      A(    ;
      A     M   2000.6;
      AN    M   2001.0;
      A     M   2010.4;
      A     M   2201.0;
      O     ;
      A     M   2000.5;
      A     DB51.DBX  608.4;
      A     DB51.DBX  603.7;
      AN    DB51.DBX  603.6;
      O     M   2001.2;
      )     ;
      A     M   2204.3;
      A     M   2208.7;
      AN    M   2204.1;
      AN    M   2242.0;
      =     M   2242.1;
NETWORK
TITLE =

      A(    ;
      A     M   2000.6;
      AN    M   2001.0;
      AN    M   2010.4;
      A     M   2201.0;
      O     ;
      A     M   2000.5;
      A     DB51.DBX  608.5;
      A     DB51.DBX  603.6;
      AN    DB51.DBX  603.7;
      )     ;
      A     M   2204.0;
      A     M   2208.7;
      AN    M   2204.2;
      AN    M   2242.3;
      =     M   2242.2;
NETWORK
TITLE =

      A(    ;
      A     M   2000.6;
      AN    M   2001.0;
      A     M   2010.4;
      A     M   2201.0;
      O     ;
      A     M   2000.5;
      A     DB51.DBX  608.5;
      A     DB51.DBX  603.7;
      AN    DB51.DBX  603.6;
      O     M   2001.2;
      )     ;
      A     M   2204.0;
      A     M   2208.7;
      AN    M   2204.3;
      AN    M   2242.2;
      =     M   2242.3;
NETWORK
TITLE =
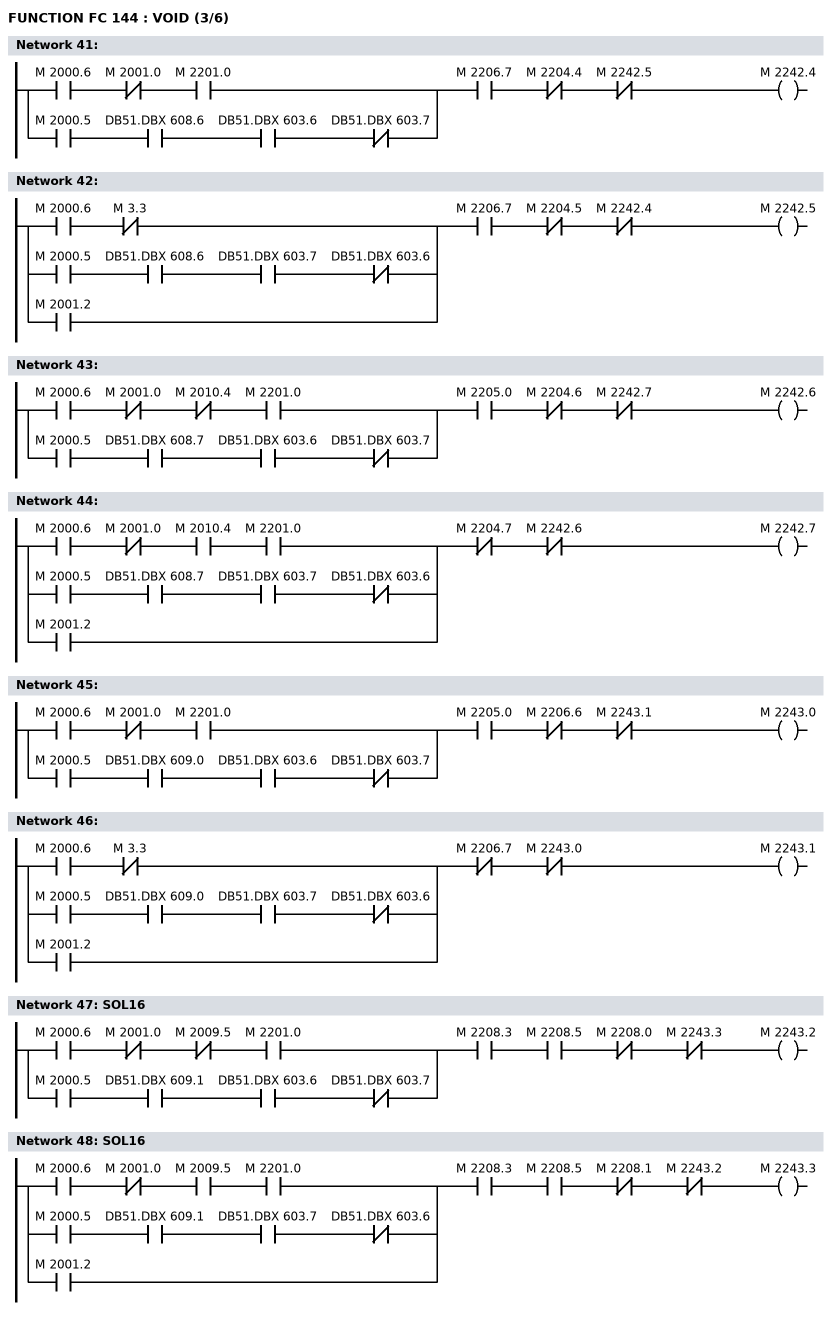

      A(    ;
      A     M   2000.6;
      AN    M   2001.0;
      A     M   2201.0;
      O     ;
      A     M   2000.5;
      A     DB51.DBX  608.6;
      A     DB51.DBX  603.6;
      AN    DB51.DBX  603.7;
      )     ;
      A     M   2206.7;
      AN    M   2204.4;
      AN    M   2242.5;
      =     M   2242.4;
NETWORK
TITLE =

      A(    ;
      A     M   2000.6;
      AN    M      3.3;
      O     ;
      A     M   2000.5;
      A     DB51.DBX  608.6;
      A     DB51.DBX  603.7;
      AN    DB51.DBX  603.6;
      O     M   2001.2;
      )     ;
      A     M   2206.7;
      AN    M   2204.5;
      AN    M   2242.4;
      =     M   2242.5;
NETWORK
TITLE =

      A(    ;
      A     M   2000.6;
      AN    M   2001.0;
      AN    M   2010.4;
      A     M   2201.0;
      O     ;
      A     M   2000.5;
      A     DB51.DBX  608.7;
      A     DB51.DBX  603.6;
      AN    DB51.DBX  603.7;
      )     ;
      A     M   2205.0;
      AN    M   2204.6;
      AN    M   2242.7;
      =     M   2242.6;
NETWORK
TITLE =

      A(    ;
      A     M   2000.6;
      AN    M   2001.0;
      A     M   2010.4;
      A     M   2201.0;
      O     ;
      A     M   2000.5;
      A     DB51.DBX  608.7;
      A     DB51.DBX  603.7;
      AN    DB51.DBX  603.6;
      O     M   2001.2;
      )     ;
      AN    M   2204.7;
      AN    M   2242.6;
      =     M   2242.7;
NETWORK
TITLE =

      A(    ;
      A     M   2000.6;
      AN    M   2001.0;
      A     M   2201.0;
      O     ;
      A     M   2000.5;
      A     DB51.DBX  609.0;
      A     DB51.DBX  603.6;
      AN    DB51.DBX  603.7;
      )     ;
      A     M   2205.0;
      AN    M   2206.6;
      AN    M   2243.1;
      =     M   2243.0;
NETWORK
TITLE =

      A(    ;
      A     M   2000.6;
      AN    M      3.3;
      O     ;
      A     M   2000.5;
      A     DB51.DBX  609.0;
      A     DB51.DBX  603.7;
      AN    DB51.DBX  603.6;
      O     M   2001.2;
      )     ;
      AN    M   2206.7;
      AN    M   2243.0;
      =     M   2243.1;
NETWORK
TITLE =SOL16

      A(    ;
      A     M   2000.6;
      AN    M   2001.0;
      AN    M   2009.5;
      A     M   2201.0;
      O     ;
      A     M   2000.5;
      A     DB51.DBX  609.1;
      A     DB51.DBX  603.6;
      AN    DB51.DBX  603.7;
      )     ;
      A     M   2208.3;
      A     M   2208.5;
      AN    M   2208.0;
      AN    M   2243.3;
      =     M   2243.2;
NETWORK
TITLE =SOL16

      A(    ;
      A     M   2000.6;
      AN    M   2001.0;
      A     M   2009.5;
      A     M   2201.0;
      O     ;
      A     M   2000.5;
      A     DB51.DBX  609.1;
      A     DB51.DBX  603.7;
      AN    DB51.DBX  603.6;
      O     M   2001.2;
      )     ;
      A     M   2208.3;
      A     M   2208.5;
      AN    M   2208.1;
      AN    M   2243.2;
      =     M   2243.3;
NETWORK
TITLE =SOL17
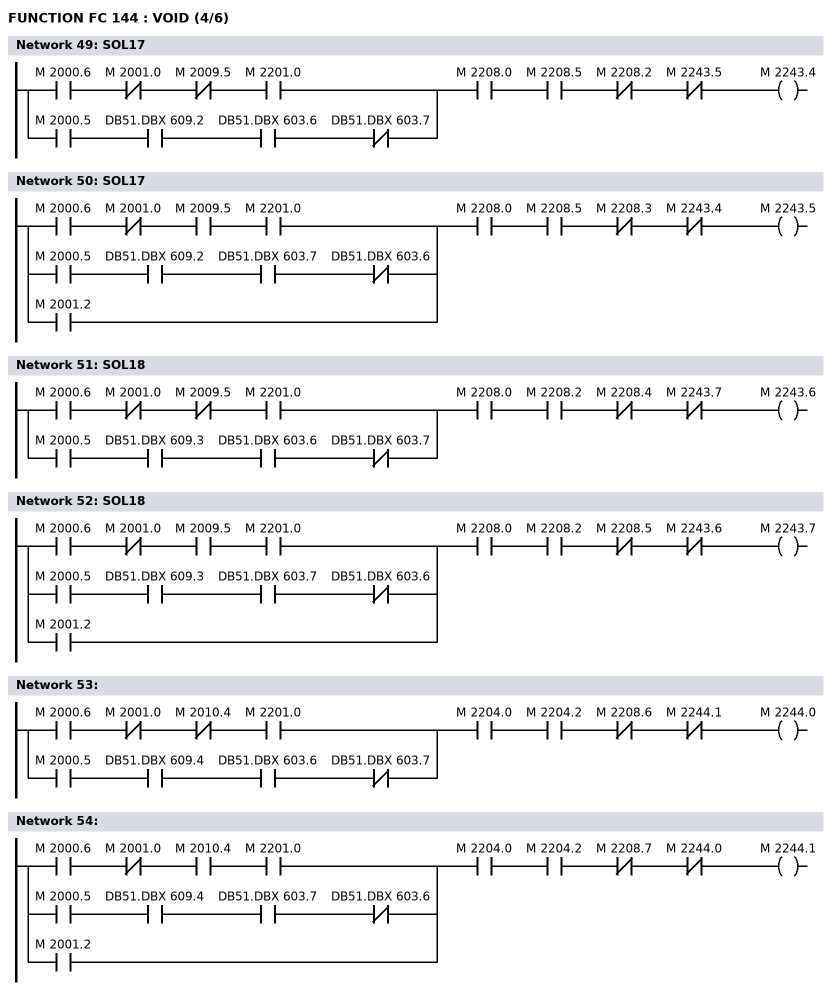

      A(    ;
      A     M   2000.6;
      AN    M   2001.0;
      AN    M   2009.5;
      A     M   2201.0;
      O     ;
      A     M   2000.5;
      A     DB51.DBX  609.2;
      A     DB51.DBX  603.6;
      AN    DB51.DBX  603.7;
      )     ;
      A     M   2208.0;
      A     M   2208.5;
      AN    M   2208.2;
      AN    M   2243.5;
      =     M   2243.4;
NETWORK
TITLE =SOL17

      A(    ;
      A     M   2000.6;
      AN    M   2001.0;
      A     M   2009.5;
      A     M   2201.0;
      O     ;
      A     M   2000.5;
      A     DB51.DBX  609.2;
      A     DB51.DBX  603.7;
      AN    DB51.DBX  603.6;
      O     M   2001.2;
      )     ;
      A     M   2208.0;
      A     M   2208.5;
      AN    M   2208.3;
      AN    M   2243.4;
      =     M   2243.5;
NETWORK
TITLE =SOL18

      A(    ;
      A     M   2000.6;
      AN    M   2001.0;
      AN    M   2009.5;
      A     M   2201.0;
      O     ;
      A     M   2000.5;
      A     DB51.DBX  609.3;
      A     DB51.DBX  603.6;
      AN    DB51.DBX  603.7;
      )     ;
      A     M   2208.0;
      A     M   2208.2;
      AN    M   2208.4;
      AN    M   2243.7;
      =     M   2243.6;
NETWORK
TITLE =SOL18

      A(    ;
      A     M   2000.6;
      AN    M   2001.0;
      A     M   2009.5;
      A     M   2201.0;
      O     ;
      A     M   2000.5;
      A     DB51.DBX  609.3;
      A     DB51.DBX  603.7;
      AN    DB51.DBX  603.6;
      O     M   2001.2;
      )     ;
      A     M   2208.0;
      A     M   2208.2;
      AN    M   2208.5;
      AN    M   2243.6;
      =     M   2243.7;
NETWORK
TITLE =

      A(    ;
      A     M   2000.6;
      AN    M   2001.0;
      AN    M   2010.4;
      A     M   2201.0;
      O     ;
      A     M   2000.5;
      A     DB51.DBX  609.4;
      A     DB51.DBX  603.6;
      AN    DB51.DBX  603.7;
      )     ;
      A     M   2204.0;
      A     M   2204.2;
      AN    M   2208.6;
      AN    M   2244.1;
      =     M   2244.0;
NETWORK
TITLE =

      A(    ;
      A     M   2000.6;
      AN    M   2001.0;
      A     M   2010.4;
      A     M   2201.0;
      O     ;
      A     M   2000.5;
      A     DB51.DBX  609.4;
      A     DB51.DBX  603.7;
      AN    DB51.DBX  603.6;
      O     M   2001.2;
      )     ;
      A     M   2204.0;
      A     M   2204.2;
      AN    M   2208.7;
      AN    M   2244.0;
      =     M   2244.1;
NETWORK
TITLE =TL 대차 SOL 동작회로
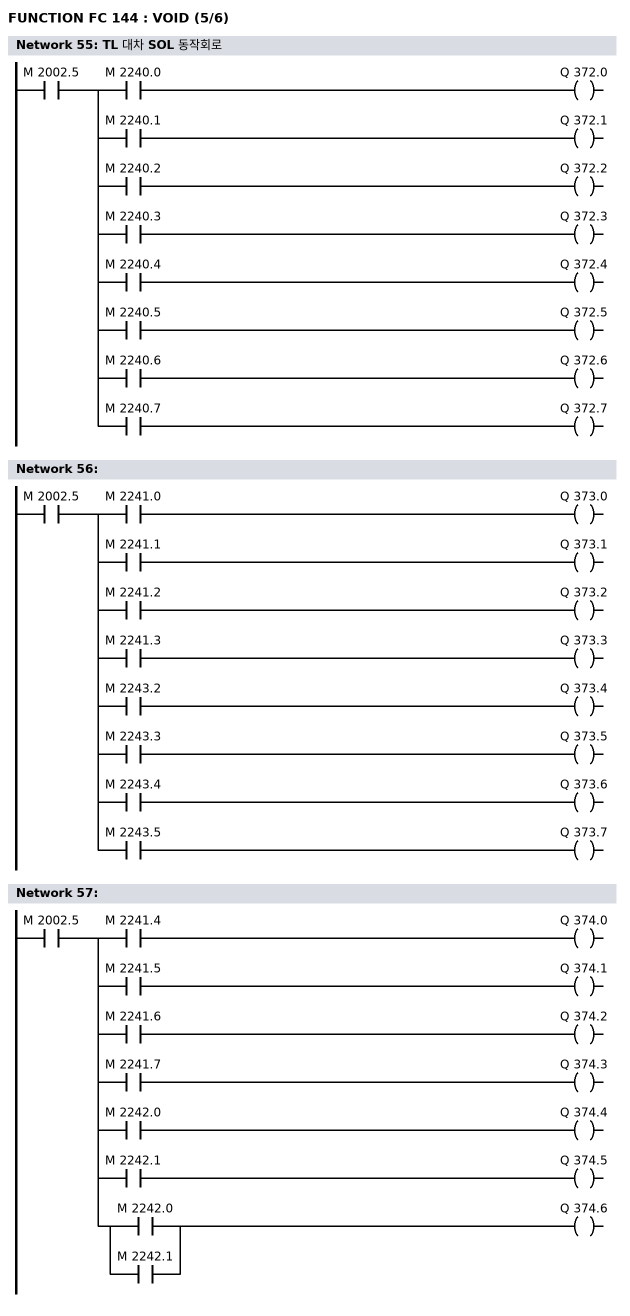

      A     M   2002.5;
      =     L      0.0;
      A     L      0.0;
      A     M   2240.0;
      =     Q    372.0;
      A     L      0.0;
      A     M   2240.1;
      =     Q    372.1;
      A     L      0.0;
      A     M   2240.2;
      =     Q    372.2;
      A     L      0.0;
      A     M   2240.3;
      =     Q    372.3;
      A     L      0.0;
      A     M   2240.4;
      =     Q    372.4;
      A     L      0.0;
      A     M   2240.5;
      =     Q    372.5;
      A     L      0.0;
      A     M   2240.6;
      =     Q    372.6;
      A     L      0.0;
      A     M   2240.7;
      =     Q    372.7;
NETWORK
TITLE =

      A     M   2002.5;
      =     L      0.0;
      A     L      0.0;
      A     M   2241.0;
      =     Q    373.0;
      A     L      0.0;
      A     M   2241.1;
      =     Q    373.1;
      A     L      0.0;
      A     M   2241.2;
      =     Q    373.2;
      A     L      0.0;
      A     M   2241.3;
      =     Q    373.3;
      A     L      0.0;
      A     M   2243.2;
      =     Q    373.4;
      A     L      0.0;
      A     M   2243.3;
      =     Q    373.5;
      A     L      0.0;
      A     M   2243.4;
      =     Q    373.6;
      A     L      0.0;
      A     M   2243.5;
      =     Q    373.7;
NETWORK
TITLE =

      A     M   2002.5;
      =     L      0.0;
      A     L      0.0;
      A     M   2241.4;
      =     Q    374.0;
      A     L      0.0;
      A     M   2241.5;
      =     Q    374.1;
      A     L      0.0;
      A     M   2241.6;
      =     Q    374.2;
      A     L      0.0;
      A     M   2241.7;
      =     Q    374.3;
      A     L      0.0;
      A     M   2242.0;
      =     Q    374.4;
      A     L      0.0;
      A     M   2242.1;
      =     Q    374.5;
      A     L      0.0;
      A(    ;
      O     M   2242.0;
      O     M   2242.1;
      )     ;
      =     Q    374.6;
NETWORK
TITLE =
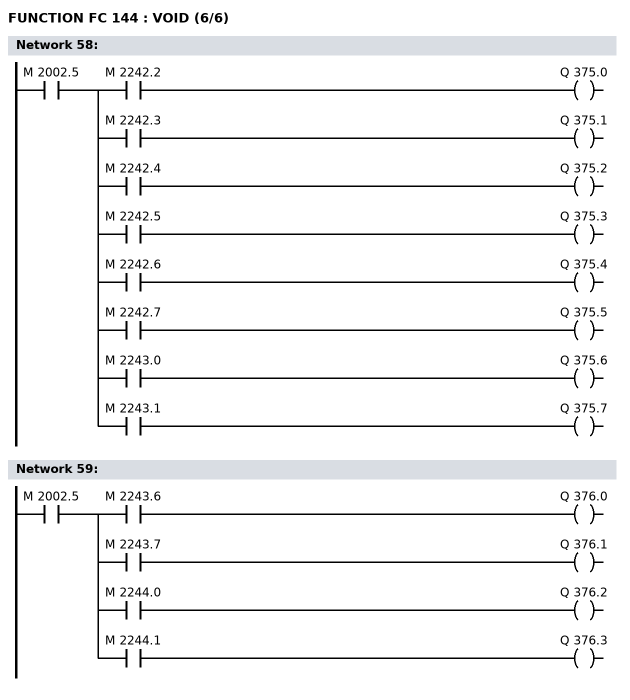

      A     M   2002.5;
      =     L      0.0;
      A     L      0.0;
      A     M   2242.2;
      =     Q    375.0;
      A     L      0.0;
      A     M   2242.3;
      =     Q    375.1;
      A     L      0.0;
      A     M   2242.4;
      =     Q    375.2;
      A     L      0.0;
      A     M   2242.5;
      =     Q    375.3;
      A     L      0.0;
      A     M   2242.6;
      =     Q    375.4;
      A     L      0.0;
      A     M   2242.7;
      =     Q    375.5;
      A     L      0.0;
      A     M   2243.0;
      =     Q    375.6;
      A     L      0.0;
      A     M   2243.1;
      =     Q    375.7;
NETWORK
TITLE =

      A     M   2002.5;
      =     L      0.0;
      A     L      0.0;
      A     M   2243.6;
      =     Q    376.0;
      A     L      0.0;
      A     M   2243.7;
      =     Q    376.1;
      A     L      0.0;
      A     M   2244.0;
      =     Q    376.2;
      A     L      0.0;
      A     M   2244.1;
      =     Q    376.3;
END_FUNCTION

FUNCTION FC 145 : VOID
TITLE =
VERSION : 0.1

BEGIN
NETWORK
TITLE =
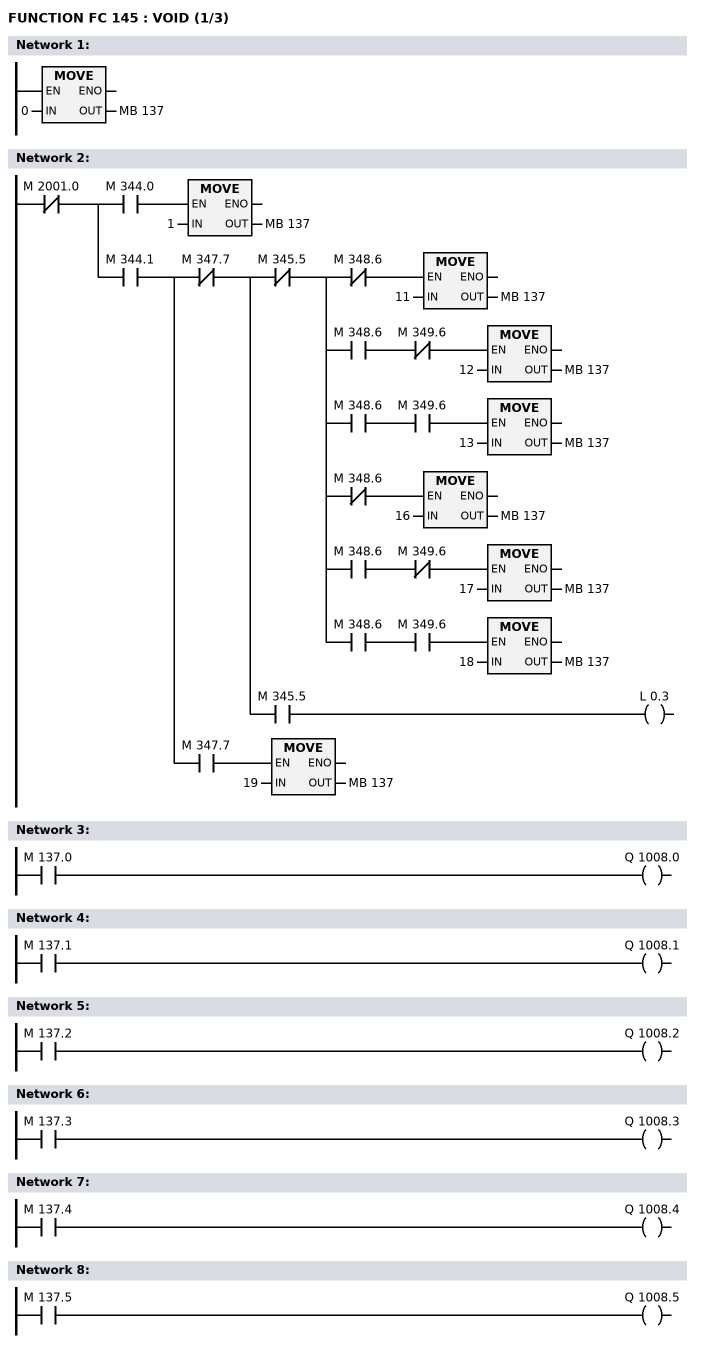

      L     0;
      T     MB   137;
      NOP   0;
NETWORK
TITLE =

      AN    M   2001.0;
      =     L      0.0;
      A     L      0.0;
      A     M    344.0;
      JNB   _001;
      L     1;
      T     MB   137;
_001: NOP   0;
      A     L      0.0;
      A     M    344.1;
      =     L      0.1;
      A     L      0.1;
      AN    M    347.7;
      =     L      0.2;
      A     L      0.2;
      AN    M    345.5;
      =     L      0.3;
      A     L      0.3;
      AN    M    348.6;
      JNB   _002;
      L     11;
      T     MB   137;
_002: NOP   0;
      A     L      0.3;
      A     M    348.6;
      AN    M    349.6;
      JNB   _003;
      L     12;
      T     MB   137;
_003: NOP   0;
      A     L      0.3;
      A     M    348.6;
      A     M    349.6;
      JNB   _004;
      L     13;
      T     MB   137;
_004: NOP   0;
      A     L      0.2;
      A     M    345.5;
      =     L      0.3;
      A     L      0.3;
      AN    M    348.6;
      JNB   _005;
      L     16;
      T     MB   137;
_005: NOP   0;
      A     L      0.3;
      A     M    348.6;
      AN    M    349.6;
      JNB   _006;
      L     17;
      T     MB   137;
_006: NOP   0;
      A     L      0.3;
      A     M    348.6;
      A     M    349.6;
      JNB   _007;
      L     18;
      T     MB   137;
_007: NOP   0;
      A     L      0.1;
      A     M    347.7;
      JNB   _008;
      L     19;
      T     MB   137;
_008: NOP   0;
NETWORK
TITLE =

      A     M    137.0;
      =     Q   1008.0;
NETWORK
TITLE =

      A     M    137.1;
      =     Q   1008.1;
NETWORK
TITLE =

      A     M    137.2;
      =     Q   1008.2;
NETWORK
TITLE =

      A     M    137.3;
      =     Q   1008.3;
NETWORK
TITLE =

      A     M    137.4;
      =     Q   1008.4;
NETWORK
TITLE =

      A     M    137.5;
      =     Q   1008.5;
NETWORK
TITLE =
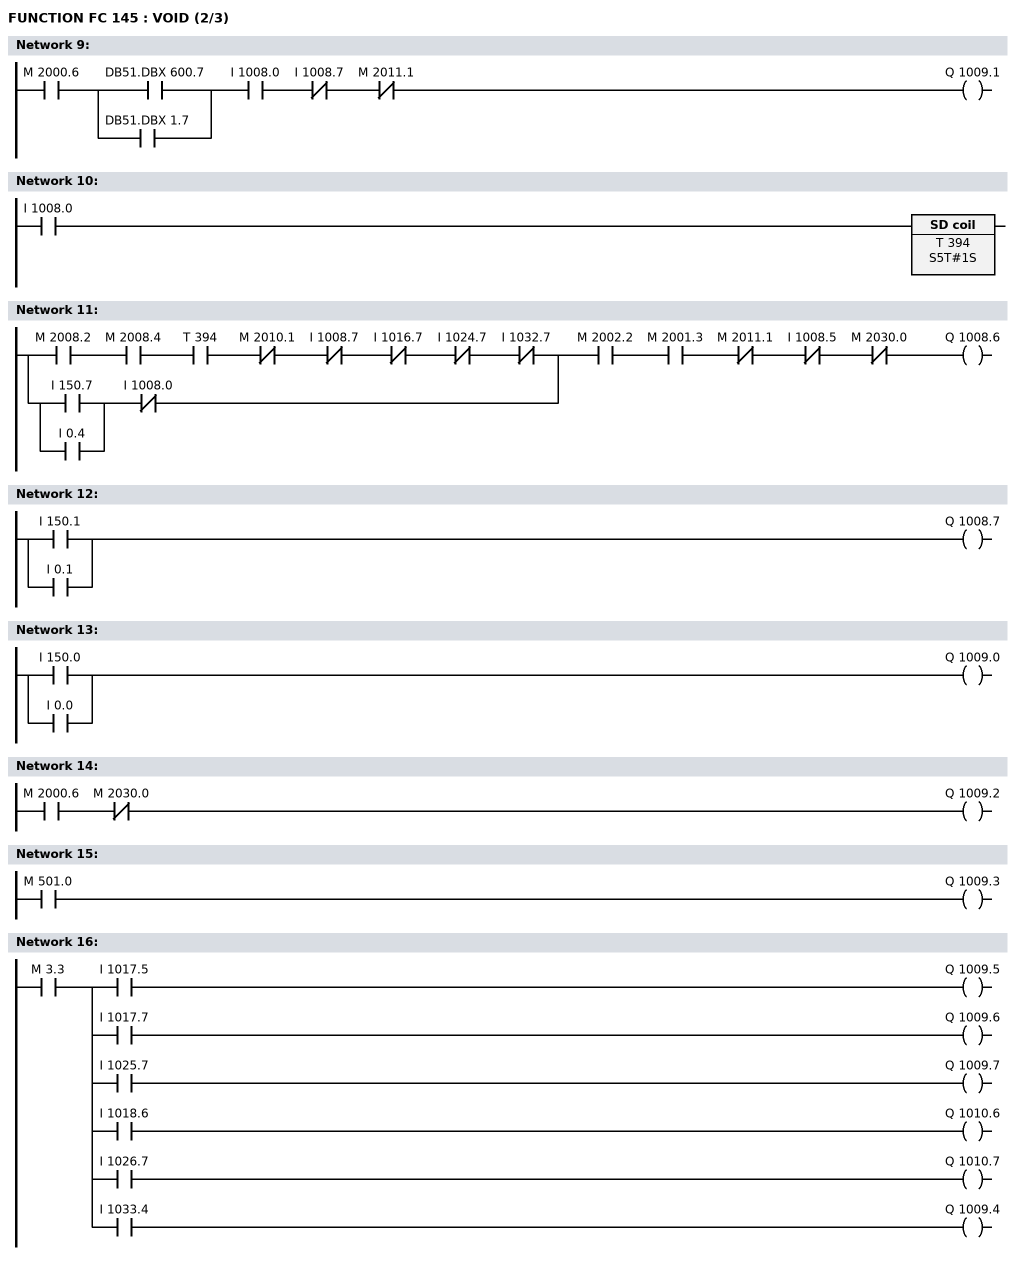

      A     M   2000.6;
      A(    ;
      O     DB51.DBX  600.7;
      O     DB51.DBX    1.7;
      )     ;
      A     I   1008.0;
      AN    I   1008.7;
      AN    M   2011.1;
      =     Q   1009.1;
NETWORK
TITLE =

      A     I   1008.0;
      L     S5T#1S;
      SD    T    394;
NETWORK
TITLE =

      A(    ;
      A     M   2008.2;
      A     M   2008.4;
      A     T    394;
      AN    M   2010.1;
      AN    I   1008.7;
      AN    I   1016.7;
      AN    I   1024.7;
      AN    I   1032.7;
      O     ;
      A(    ;
      O     I    150.7;
      O     I      0.4;
      )     ;
      AN    I   1008.0;
      )     ;
      A     M   2002.2;
      A     M   2001.3;
      AN    M   2011.1;
      AN    I   1008.5;
      AN    M   2030.0;
      =     Q   1008.6;
NETWORK
TITLE =

      O     I    150.1;
      O     I      0.1;
      =     Q   1008.7;
NETWORK
TITLE =

      O     I    150.0;
      O     I      0.0;
      =     Q   1009.0;
NETWORK
TITLE =

      A     M   2000.6;
      AN    M   2030.0;
      =     Q   1009.2;
NETWORK
TITLE =

      A     M    501.0;
      =     Q   1009.3;
NETWORK
TITLE =

      A     M      3.3;
      =     L      0.0;
      A     L      0.0;
      A     I   1017.5;
      =     Q   1009.5;
      A     L      0.0;
      A     I   1017.7;
      =     Q   1009.6;
      A     L      0.0;
      A     I   1025.7;
      =     Q   1009.7;
      A     L      0.0;
      A     I   1018.6;
      =     Q   1010.6;
      A     L      0.0;
      A     I   1026.7;
      =     Q   1010.7;
      A     L      0.0;
      A     I   1033.4;
      =     Q   1009.4;
NETWORK
TITLE =
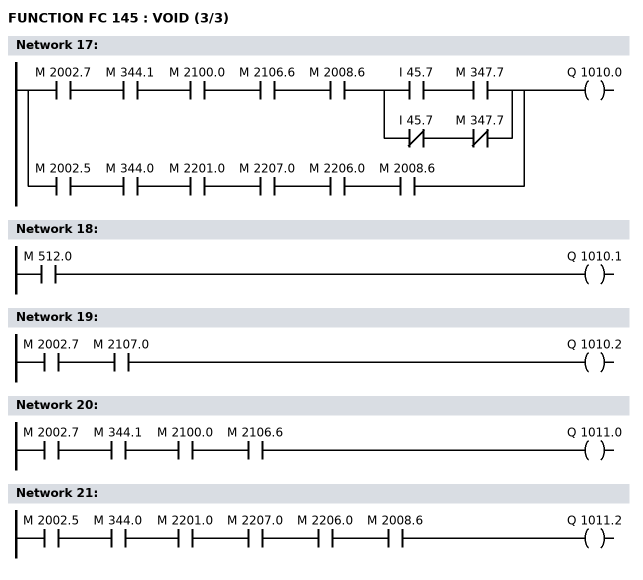

      A     M   2002.7;
      A     M    344.1;
      A     M   2100.0;
      A     M   2106.6;
      A     M   2008.6;
      A(    ;
      A     I     45.7;
      A     M    347.7;
      O     ;
      AN    I     45.7;
      AN    M    347.7;
      )     ;
      O     ;
      A     M   2002.5;
      A     M    344.0;
      A     M   2201.0;
      A     M   2207.0;
      A     M   2206.0;
      A     M   2008.6;
      =     Q   1010.0;
NETWORK
TITLE =

      A     M    512.0;
      =     Q   1010.1;
NETWORK
TITLE =

      A     M   2002.7;
      A     M   2107.0;
      =     Q   1010.2;
NETWORK
TITLE =

      A     M   2002.7;
      A     M    344.1;
      A     M   2100.0;
      A     M   2106.6;
      =     Q   1011.0;
NETWORK
TITLE =

      A     M   2002.5;
      A     M    344.0;
      A     M   2201.0;
      A     M   2207.0;
      A     M   2206.0;
      A     M   2008.6;
      =     Q   1011.2;
END_FUNCTION

FUNCTION FC 146 : VOID
TITLE =
VERSION : 0.1

BEGIN
NETWORK
TITLE =
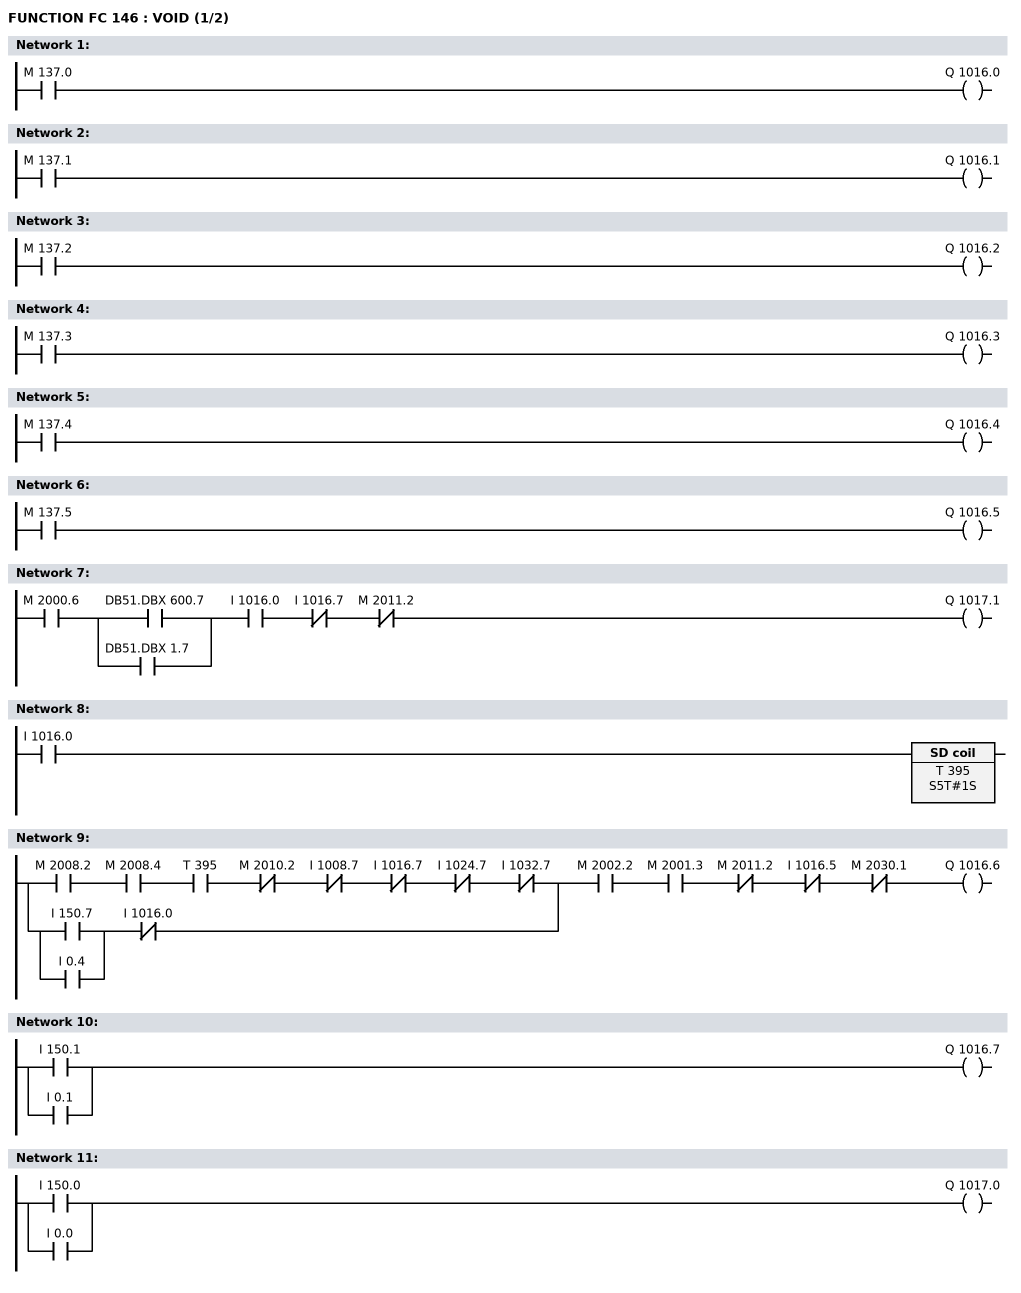

      A     M    137.0;
      =     Q   1016.0;
NETWORK
TITLE =

      A     M    137.1;
      =     Q   1016.1;
NETWORK
TITLE =

      A     M    137.2;
      =     Q   1016.2;
NETWORK
TITLE =

      A     M    137.3;
      =     Q   1016.3;
NETWORK
TITLE =

      A     M    137.4;
      =     Q   1016.4;
NETWORK
TITLE =

      A     M    137.5;
      =     Q   1016.5;
NETWORK
TITLE =

      A     M   2000.6;
      A(    ;
      O     DB51.DBX  600.7;
      O     DB51.DBX    1.7;
      )     ;
      A     I   1016.0;
      AN    I   1016.7;
      AN    M   2011.2;
      =     Q   1017.1;
NETWORK
TITLE =

      A     I   1016.0;
      L     S5T#1S;
      SD    T    395;
NETWORK
TITLE =

      A(    ;
      A     M   2008.2;
      A     M   2008.4;
      A     T    395;
      AN    M   2010.2;
      AN    I   1008.7;
      AN    I   1016.7;
      AN    I   1024.7;
      AN    I   1032.7;
      O     ;
      A(    ;
      O     I    150.7;
      O     I      0.4;
      )     ;
      AN    I   1016.0;
      )     ;
      A     M   2002.2;
      A     M   2001.3;
      AN    M   2011.2;
      AN    I   1016.5;
      AN    M   2030.1;
      =     Q   1016.6;
NETWORK
TITLE =

      O     I    150.1;
      O     I      0.1;
      =     Q   1016.7;
NETWORK
TITLE =

      O     I    150.0;
      O     I      0.0;
      =     Q   1017.0;
NETWORK
TITLE =
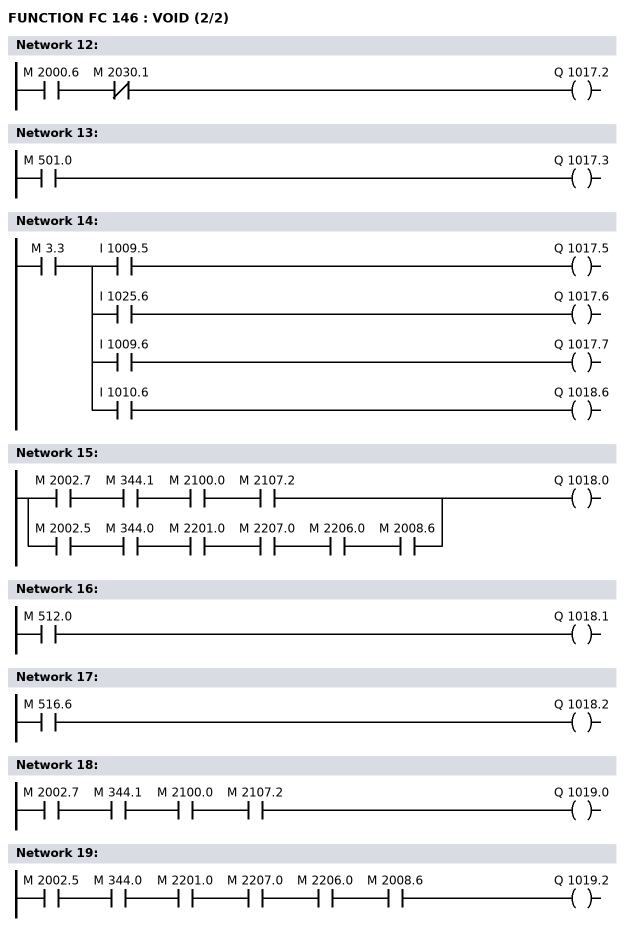

      A     M   2000.6;
      AN    M   2030.1;
      =     Q   1017.2;
NETWORK
TITLE =

      A     M    501.0;
      =     Q   1017.3;
NETWORK
TITLE =

      A     M      3.3;
      =     L      0.0;
      A     L      0.0;
      A     I   1009.5;
      =     Q   1017.5;
      A     L      0.0;
      A     I   1025.6;
      =     Q   1017.6;
      A     L      0.0;
      A     I   1009.6;
      =     Q   1017.7;
      A     L      0.0;
      A     I   1010.6;
      =     Q   1018.6;
NETWORK
TITLE =

      A     M   2002.7;
      A     M    344.1;
      A     M   2100.0;
      A     M   2107.2;
      O     ;
      A     M   2002.5;
      A     M    344.0;
      A     M   2201.0;
      A     M   2207.0;
      A     M   2206.0;
      A     M   2008.6;
      =     Q   1018.0;
NETWORK
TITLE =

      A     M    512.0;
      =     Q   1018.1;
NETWORK
TITLE =

      A     M    516.6;
      =     Q   1018.2;
NETWORK
TITLE =

      A     M   2002.7;
      A     M    344.1;
      A     M   2100.0;
      A     M   2107.2;
      =     Q   1019.0;
NETWORK
TITLE =

      A     M   2002.5;
      A     M    344.0;
      A     M   2201.0;
      A     M   2207.0;
      A     M   2206.0;
      A     M   2008.6;
      =     Q   1019.2;
END_FUNCTION

FUNCTION FC 147 : VOID
TITLE =
VERSION : 0.1

BEGIN
NETWORK
TITLE =
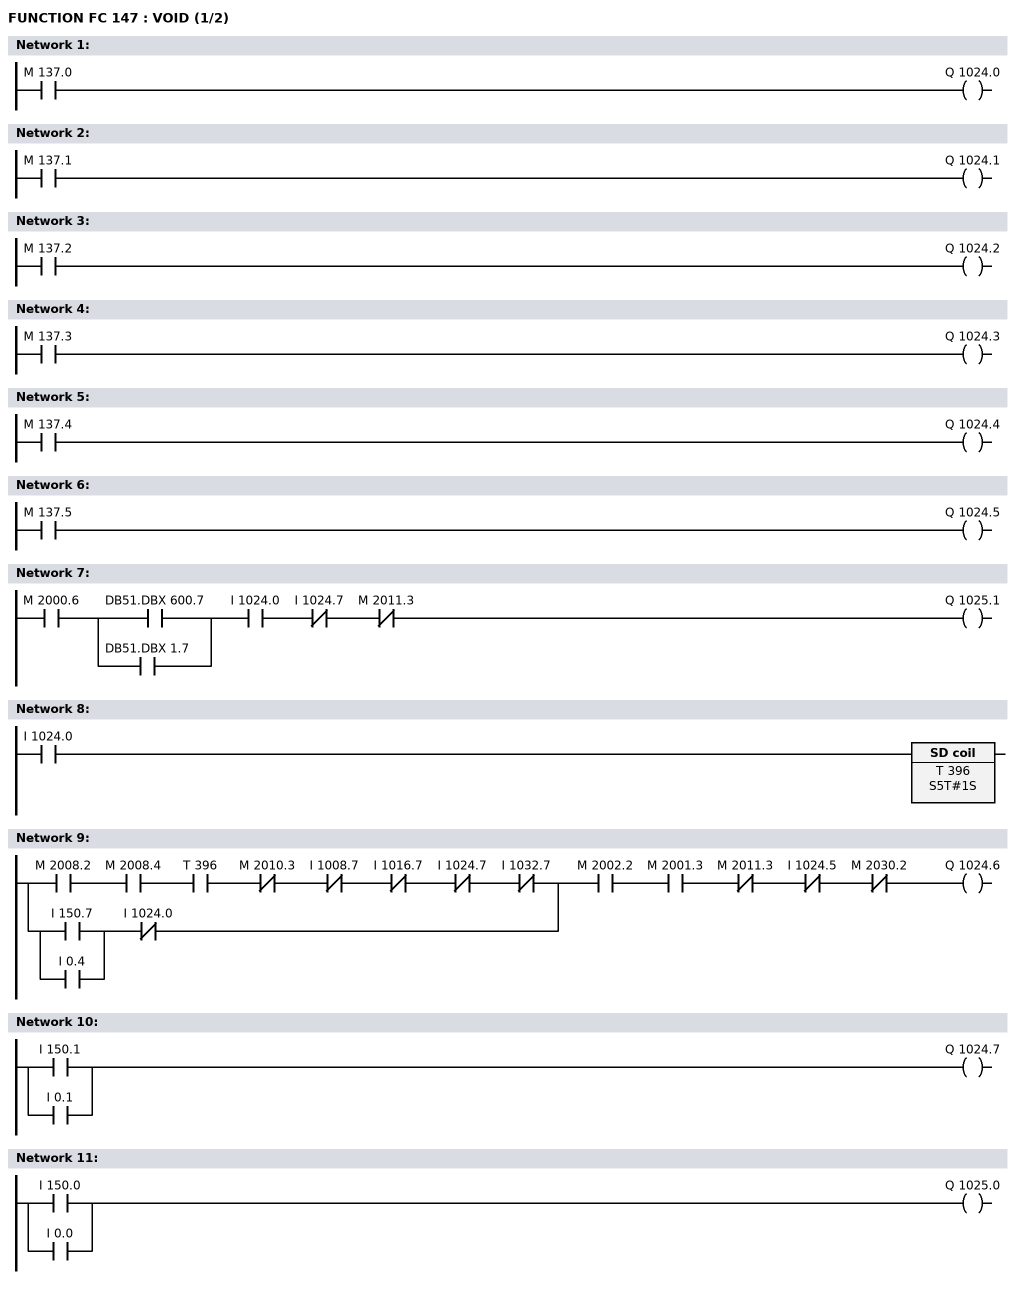

      A     M    137.0;
      =     Q   1024.0;
NETWORK
TITLE =

      A     M    137.1;
      =     Q   1024.1;
NETWORK
TITLE =

      A     M    137.2;
      =     Q   1024.2;
NETWORK
TITLE =

      A     M    137.3;
      =     Q   1024.3;
NETWORK
TITLE =

      A     M    137.4;
      =     Q   1024.4;
NETWORK
TITLE =

      A     M    137.5;
      =     Q   1024.5;
NETWORK
TITLE =

      A     M   2000.6;
      A(    ;
      O     DB51.DBX  600.7;
      O     DB51.DBX    1.7;
      )     ;
      A     I   1024.0;
      AN    I   1024.7;
      AN    M   2011.3;
      =     Q   1025.1;
NETWORK
TITLE =

      A     I   1024.0;
      L     S5T#1S;
      SD    T    396;
NETWORK
TITLE =

      A(    ;
      A     M   2008.2;
      A     M   2008.4;
      A     T    396;
      AN    M   2010.3;
      AN    I   1008.7;
      AN    I   1016.7;
      AN    I   1024.7;
      AN    I   1032.7;
      O     ;
      A(    ;
      O     I    150.7;
      O     I      0.4;
      )     ;
      AN    I   1024.0;
      )     ;
      A     M   2002.2;
      A     M   2001.3;
      AN    M   2011.3;
      AN    I   1024.5;
      AN    M   2030.2;
      =     Q   1024.6;
NETWORK
TITLE =

      O     I    150.1;
      O     I      0.1;
      =     Q   1024.7;
NETWORK
TITLE =

      O     I    150.0;
      O     I      0.0;
      =     Q   1025.0;
NETWORK
TITLE =
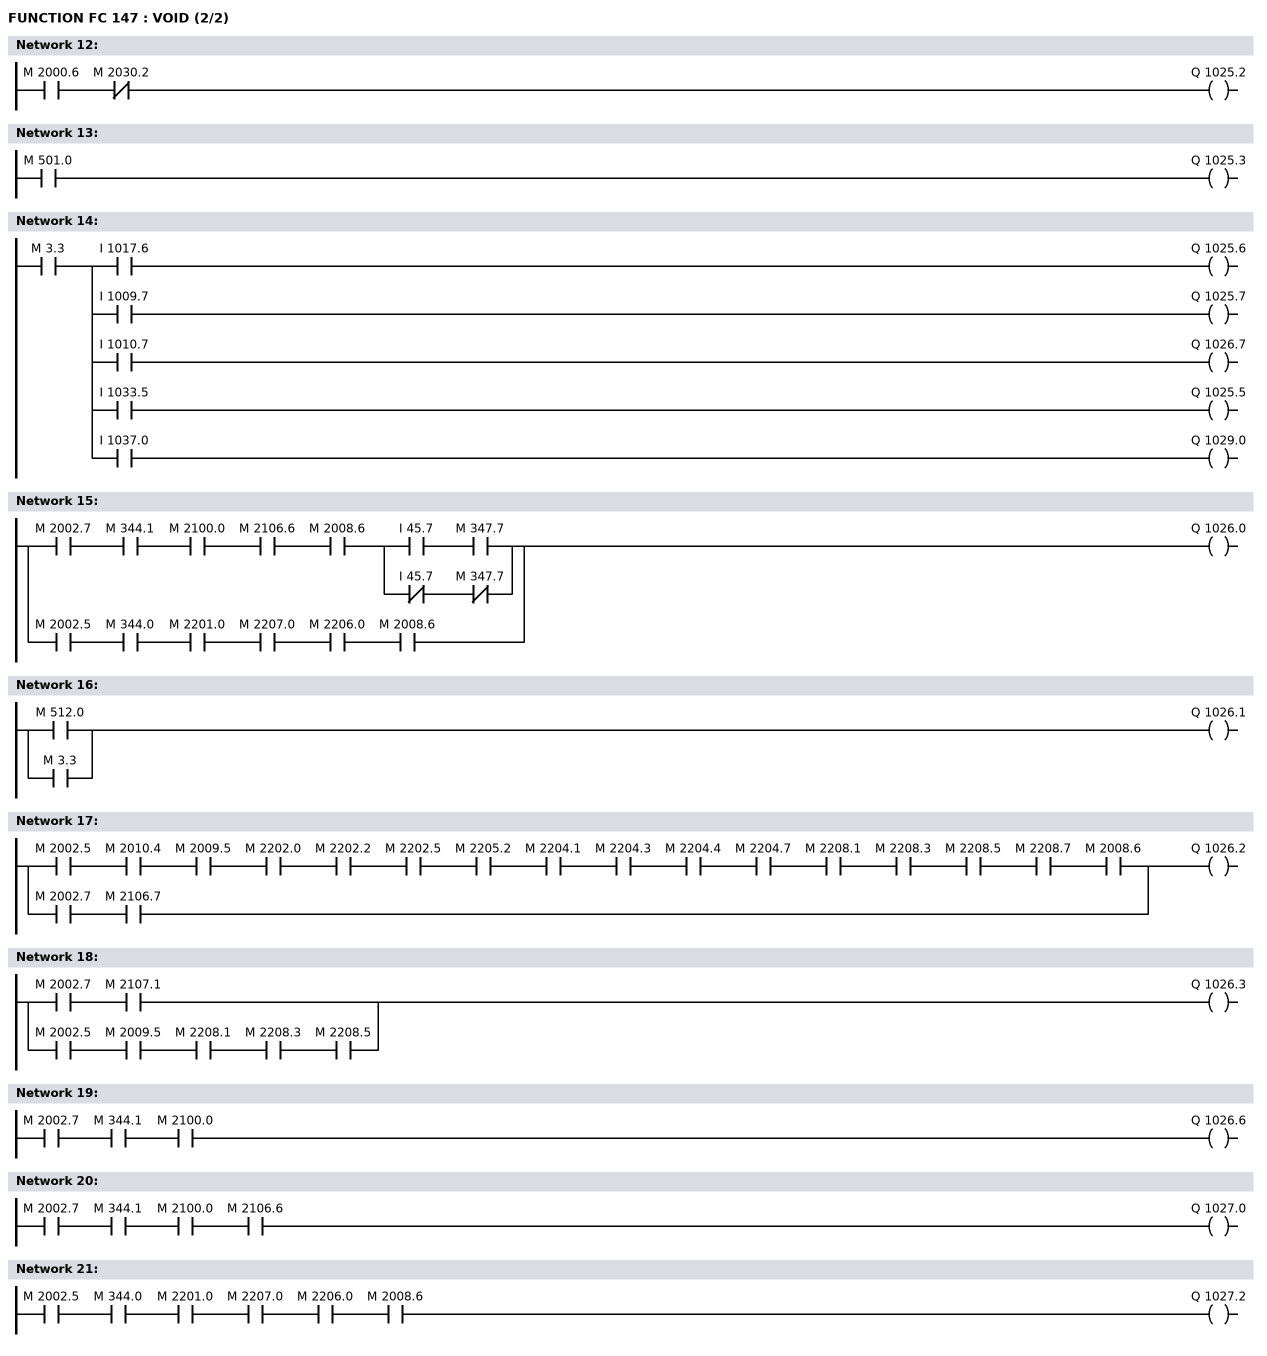

      A     M   2000.6;
      AN    M   2030.2;
      =     Q   1025.2;
NETWORK
TITLE =

      A     M    501.0;
      =     Q   1025.3;
NETWORK
TITLE =

      A     M      3.3;
      =     L      0.0;
      A     L      0.0;
      A     I   1017.6;
      =     Q   1025.6;
      A     L      0.0;
      A     I   1009.7;
      =     Q   1025.7;
      A     L      0.0;
      A     I   1010.7;
      =     Q   1026.7;
      A     L      0.0;
      A     I   1033.5;
      =     Q   1025.5;
      A     L      0.0;
      A     I   1037.0;
      =     Q   1029.0;
NETWORK
TITLE =

      A     M   2002.7;
      A     M    344.1;
      A     M   2100.0;
      A     M   2106.6;
      A     M   2008.6;
      A(    ;
      A     I     45.7;
      A     M    347.7;
      O     ;
      AN    I     45.7;
      AN    M    347.7;
      )     ;
      O     ;
      A     M   2002.5;
      A     M    344.0;
      A     M   2201.0;
      A     M   2207.0;
      A     M   2206.0;
      A     M   2008.6;
      =     Q   1026.0;
NETWORK
TITLE =

      O     M    512.0;
      O     M      3.3;
      =     Q   1026.1;
NETWORK
TITLE =

      A     M   2002.5;
      A     M   2010.4;
      A     M   2009.5;
      A     M   2202.0;
      A     M   2202.2;
      A     M   2202.5;
      A     M   2205.2;
      A     M   2204.1;
      A     M   2204.3;
      A     M   2204.4;
      A     M   2204.7;
      A     M   2208.1;
      A     M   2208.3;
      A     M   2208.5;
      A     M   2208.7;
      A     M   2008.6;
      O     ;
      A     M   2002.7;
      A     M   2106.7;
      =     Q   1026.2;
NETWORK
TITLE =

      A     M   2002.7;
      A     M   2107.1;
      O     ;
      A     M   2002.5;
      A     M   2009.5;
      A     M   2208.1;
      A     M   2208.3;
      A     M   2208.5;
      =     Q   1026.3;
NETWORK
TITLE =

      A     M   2002.7;
      A     M    344.1;
      A     M   2100.0;
      =     Q   1026.6;
NETWORK
TITLE =

      A     M   2002.7;
      A     M    344.1;
      A     M   2100.0;
      A     M   2106.6;
      =     Q   1027.0;
NETWORK
TITLE =

      A     M   2002.5;
      A     M    344.0;
      A     M   2201.0;
      A     M   2207.0;
      A     M   2206.0;
      A     M   2008.6;
      =     Q   1027.2;
END_FUNCTION

FUNCTION FC 148 : VOID
TITLE =
VERSION : 0.1

BEGIN
NETWORK
TITLE =
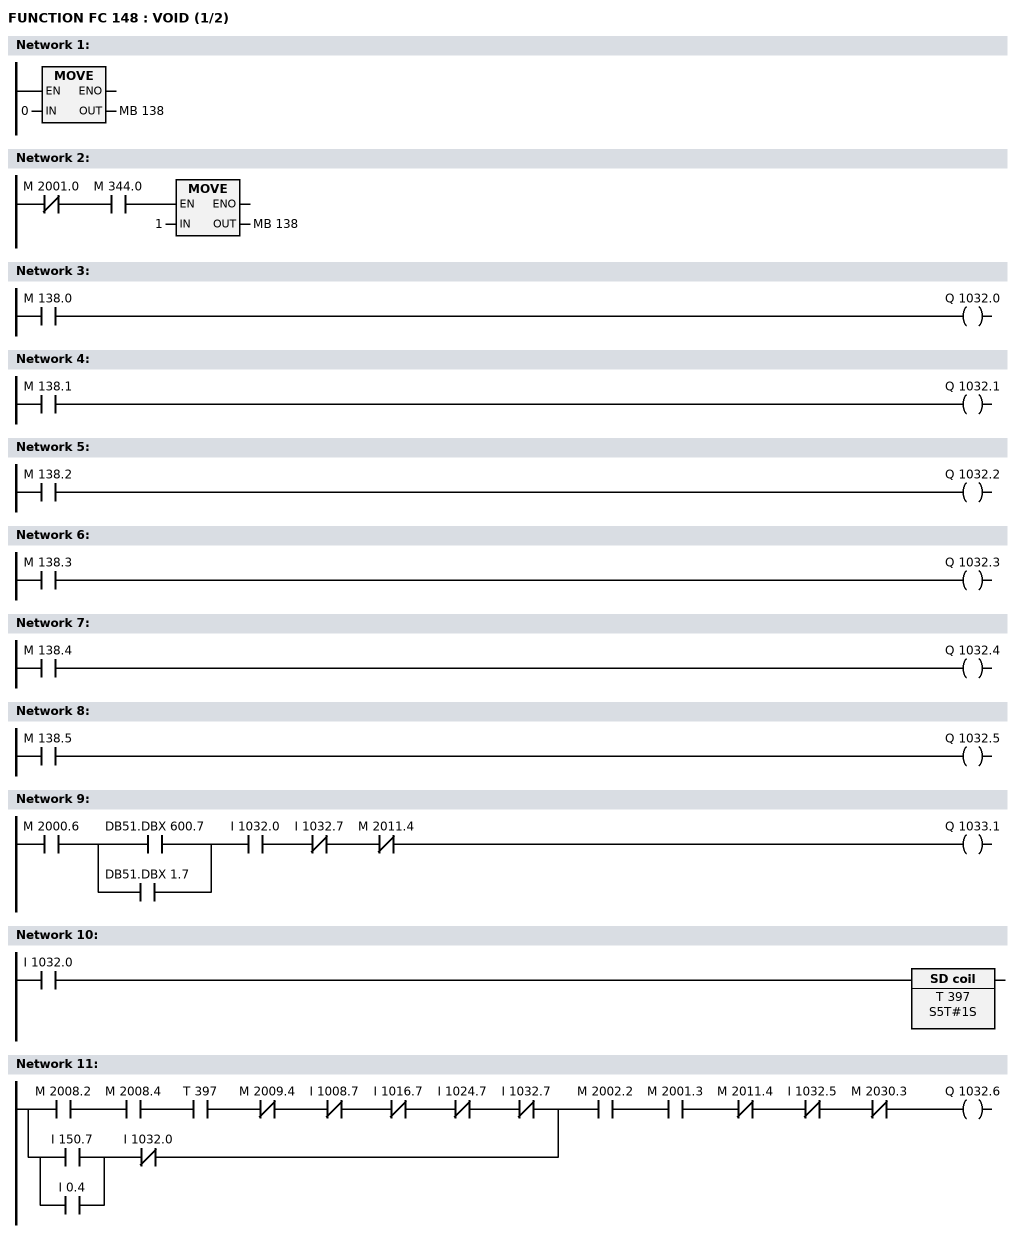

      L     0;
      T     MB   138;
      NOP   0;
NETWORK
TITLE =

      AN    M   2001.0;
      A     M    344.0;
      JNB   _001;
      L     1;
      T     MB   138;
_001: NOP   0;
NETWORK
TITLE =

      A     M    138.0;
      =     Q   1032.0;
NETWORK
TITLE =

      A     M    138.1;
      =     Q   1032.1;
NETWORK
TITLE =

      A     M    138.2;
      =     Q   1032.2;
NETWORK
TITLE =

      A     M    138.3;
      =     Q   1032.3;
NETWORK
TITLE =

      A     M    138.4;
      =     Q   1032.4;
NETWORK
TITLE =

      A     M    138.5;
      =     Q   1032.5;
NETWORK
TITLE =

      A     M   2000.6;
      A(    ;
      O     DB51.DBX  600.7;
      O     DB51.DBX    1.7;
      )     ;
      A     I   1032.0;
      AN    I   1032.7;
      AN    M   2011.4;
      =     Q   1033.1;
NETWORK
TITLE =

      A     I   1032.0;
      L     S5T#1S;
      SD    T    397;
NETWORK
TITLE =

      A(    ;
      A     M   2008.2;
      A     M   2008.4;
      A     T    397;
      AN    M   2009.4;
      AN    I   1008.7;
      AN    I   1016.7;
      AN    I   1024.7;
      AN    I   1032.7;
      O     ;
      A(    ;
      O     I    150.7;
      O     I      0.4;
      )     ;
      AN    I   1032.0;
      )     ;
      A     M   2002.2;
      A     M   2001.3;
      AN    M   2011.4;
      AN    I   1032.5;
      AN    M   2030.3;
      =     Q   1032.6;
NETWORK
TITLE =
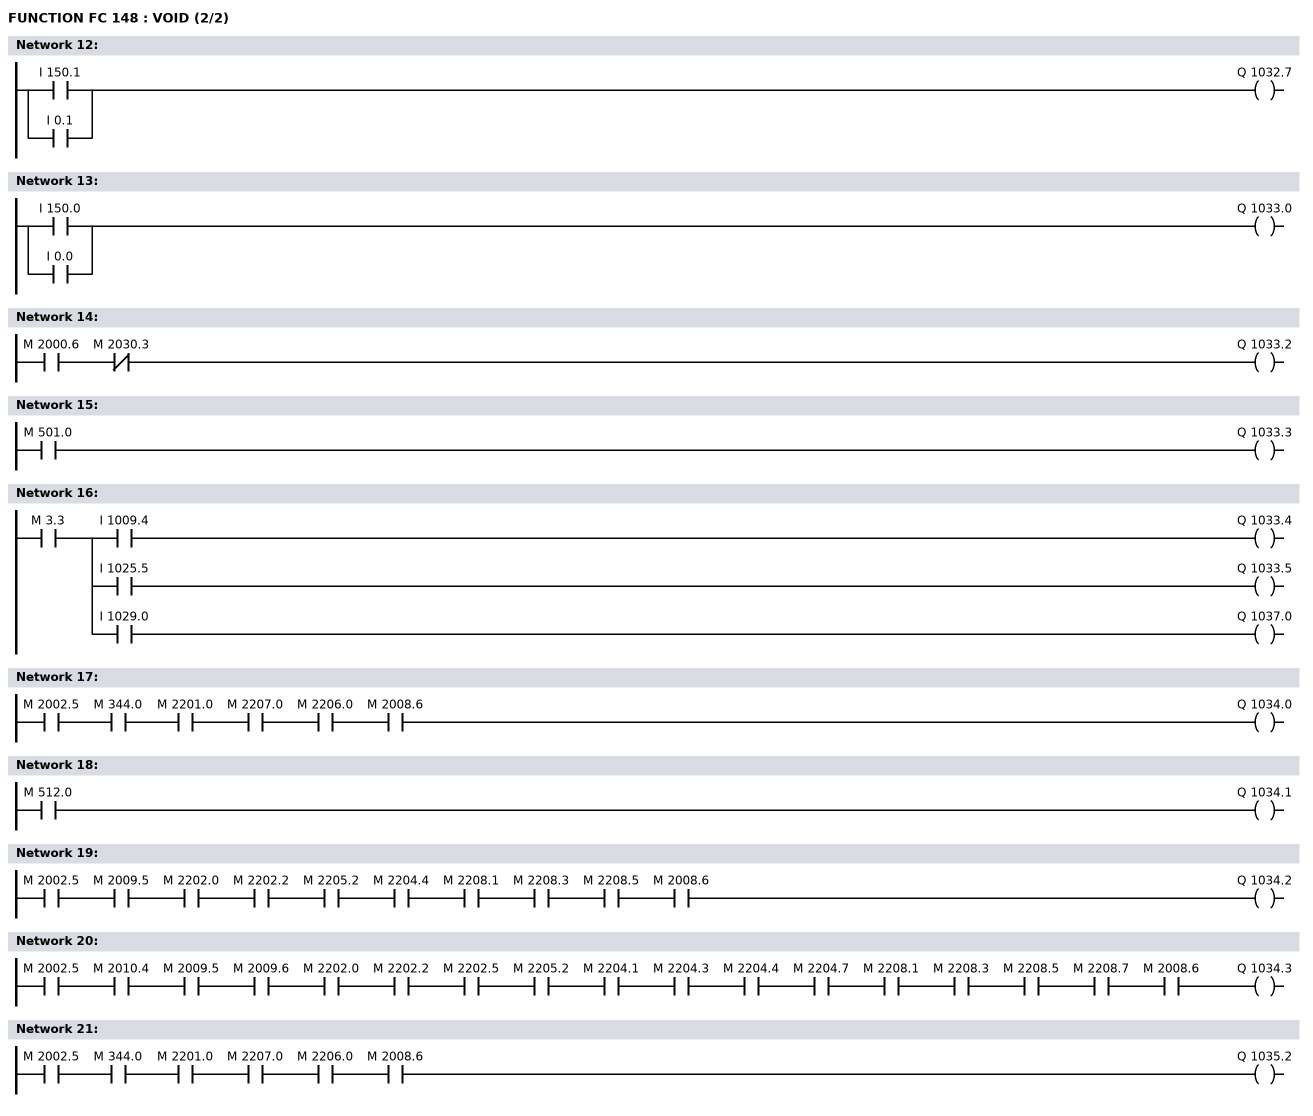

      O     I    150.1;
      O     I      0.1;
      =     Q   1032.7;
NETWORK
TITLE =

      O     I    150.0;
      O     I      0.0;
      =     Q   1033.0;
NETWORK
TITLE =

      A     M   2000.6;
      AN    M   2030.3;
      =     Q   1033.2;
NETWORK
TITLE =

      A     M    501.0;
      =     Q   1033.3;
NETWORK
TITLE =

      A     M      3.3;
      =     L      0.0;
      A     L      0.0;
      A     I   1009.4;
      =     Q   1033.4;
      A     L      0.0;
      A     I   1025.5;
      =     Q   1033.5;
      A     L      0.0;
      A     I   1029.0;
      =     Q   1037.0;
NETWORK
TITLE =

      A     M   2002.5;
      A     M    344.0;
      A     M   2201.0;
      A     M   2207.0;
      A     M   2206.0;
      A     M   2008.6;
      =     Q   1034.0;
NETWORK
TITLE =

      A     M    512.0;
      =     Q   1034.1;
NETWORK
TITLE =

      A     M   2002.5;
      A     M   2009.5;
      A     M   2202.0;
      A     M   2202.2;
      A     M   2205.2;
      A     M   2204.4;
      A     M   2208.1;
      A     M   2208.3;
      A     M   2208.5;
      A     M   2008.6;
      =     Q   1034.2;
NETWORK
TITLE =

      A     M   2002.5;
      A     M   2010.4;
      A     M   2009.5;
      A     M   2009.6;
      A     M   2202.0;
      A     M   2202.2;
      A     M   2202.5;
      A     M   2205.2;
      A     M   2204.1;
      A     M   2204.3;
      A     M   2204.4;
      A     M   2204.7;
      A     M   2208.1;
      A     M   2208.3;
      A     M   2208.5;
      A     M   2208.7;
      A     M   2008.6;
      =     Q   1034.3;
NETWORK
TITLE =

      A     M   2002.5;
      A     M    344.0;
      A     M   2201.0;
      A     M   2207.0;
      A     M   2206.0;
      A     M   2008.6;
      =     Q   1035.2;
END_FUNCTION

FUNCTION_BLOCK FB 150
TITLE =
VERSION : 0.1


VAR
  S_DOWN_DL_MODE : FB 402;
END_VAR
BEGIN
NETWORK
TITLE =
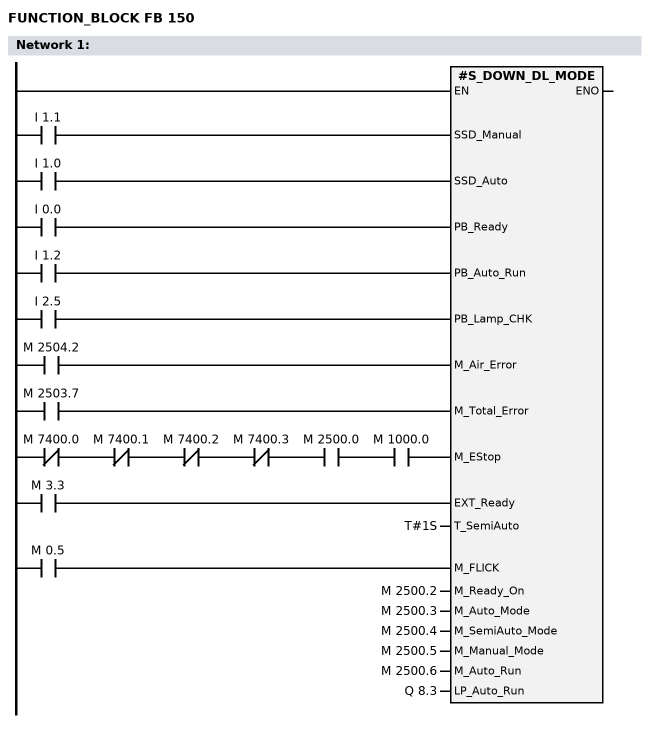

      A     I      1.1;
      =     L      0.0;
      BLD   103;
      A     I      1.0;
      =     L      0.1;
      BLD   103;
      A     I      0.0;
      =     L      0.2;
      BLD   103;
      A     I      1.2;
      =     L      0.3;
      BLD   103;
      A     I      2.5;
      =     L      0.6;
      BLD   103;
      A     M   2504.2;
      =     L      0.7;
      BLD   103;
      A     M   2503.7;
      =     L      1.1;
      BLD   103;
      AN    M   7400.0;
      AN    M   7400.1;
      AN    M   7400.2;
      AN    M   7400.3;
      A     M   2500.0;
      A     M   1000.0;
      =     L      1.2;
      BLD   103;
      A     M      3.3;
      =     L      1.3;
      BLD   103;
      A     M      0.5;
      =     L      1.5;
      BLD   103;
      CALL #S_DOWN_DL_MODE (
           SSD_Manual               := L      0.0,
           SSD_Auto                 := L      0.1,
           PB_Ready                 := L      0.2,
           PB_Auto_Run              := L      0.3,
           PB_Lamp_CHK              := L      0.6,
           M_Air_Error              := L      0.7,
           M_Total_Error            := L      1.1,
           M_EStop                  := L      1.2,
           EXT_Ready                := L      1.3,
           T_SemiAuto               := T#1S,
           M_FLICK                  := L      1.5,
           M_Ready_On               := M   2500.2,
           M_Auto_Mode              := M   2500.3,
           M_SemiAuto_Mode          := M   2500.4,
           M_Manual_Mode            := M   2500.5,
           M_Auto_Run               := M   2500.6,
           LP_Auto_Run              := Q      8.3);
      NOP   0;
END_FUNCTION_BLOCK

DATA_BLOCK DB 150
TITLE =
VERSION : 0.0

 FB 150
BEGIN
   S_DOWN_DL_MODE.SSD_Manual := FALSE;
   S_DOWN_DL_MODE.SSD_Auto := FALSE;
   S_DOWN_DL_MODE.PB_Ready := FALSE;
   S_DOWN_DL_MODE.PB_Auto_Run := FALSE;
   S_DOWN_DL_MODE.PB_Remote_Ready := FALSE;
   S_DOWN_DL_MODE.PB_Remote_Auto_Run := FALSE;
   S_DOWN_DL_MODE.PB_Lamp_CHK := FALSE;
   S_DOWN_DL_MODE.M_Air_Error := FALSE;
   S_DOWN_DL_MODE.M_Water_Error := FALSE;
   S_DOWN_DL_MODE.M_Total_Error := FALSE;
   S_DOWN_DL_MODE.M_EStop := FALSE;
   S_DOWN_DL_MODE.EXT_Ready := FALSE;
   S_DOWN_DL_MODE.EXT_Auto := FALSE;
   S_DOWN_DL_MODE.T_SemiAuto := T#0MS;
   S_DOWN_DL_MODE.M_FLICK := FALSE;
   S_DOWN_DL_MODE.M_Ready_On := FALSE;
   S_DOWN_DL_MODE.M_Auto_Mode := FALSE;
   S_DOWN_DL_MODE.M_SemiAuto_Mode := FALSE;
   S_DOWN_DL_MODE.M_Manual_Mode := FALSE;
   S_DOWN_DL_MODE.M_Auto_Run := FALSE;
   S_DOWN_DL_MODE.LP_Ready_On := FALSE;
   S_DOWN_DL_MODE.LP_Auto_Run := FALSE;
   S_DOWN_DL_MODE.AUTO_MODE_DELAY.IN := FALSE;
   S_DOWN_DL_MODE.AUTO_MODE_DELAY.PT := T#0MS;
   S_DOWN_DL_MODE.AUTO_MODE_DELAY.Q := FALSE;
   S_DOWN_DL_MODE.AUTO_MODE_DELAY.ET := T#0MS;
   S_DOWN_DL_MODE.AUTO_MODE_DELAY.STATE := B#16#0;
   S_DOWN_DL_MODE.AUTO_MODE_DELAY.STIME := T#0MS;
   S_DOWN_DL_MODE.AUTO_MODE_DELAY.ATIME := T#0MS;
   S_DOWN_DL_MODE.SEMI_AUTO_DELAY.IN := FALSE;
   S_DOWN_DL_MODE.SEMI_AUTO_DELAY.PT := T#0MS;
   S_DOWN_DL_MODE.SEMI_AUTO_DELAY.Q := FALSE;
   S_DOWN_DL_MODE.SEMI_AUTO_DELAY.ET := T#0MS;
   S_DOWN_DL_MODE.SEMI_AUTO_DELAY.STATE := B#16#0;
   S_DOWN_DL_MODE.SEMI_AUTO_DELAY.STIME := T#0MS;
   S_DOWN_DL_MODE.SEMI_AUTO_DELAY.ATIME := T#0MS;
   S_DOWN_DL_MODE.MANUAL_DELAY.IN := FALSE;
   S_DOWN_DL_MODE.MANUAL_DELAY.PT := T#0MS;
   S_DOWN_DL_MODE.MANUAL_DELAY.Q := FALSE;
   S_DOWN_DL_MODE.MANUAL_DELAY.ET := T#0MS;
   S_DOWN_DL_MODE.MANUAL_DELAY.STATE := B#16#0;
   S_DOWN_DL_MODE.MANUAL_DELAY.STIME := T#0MS;
   S_DOWN_DL_MODE.MANUAL_DELAY.ATIME := T#0MS;
END_DATA_BLOCK

FUNCTION FC 150 : VOID
TITLE =
VERSION : 0.1

BEGIN
NETWORK
TITLE =
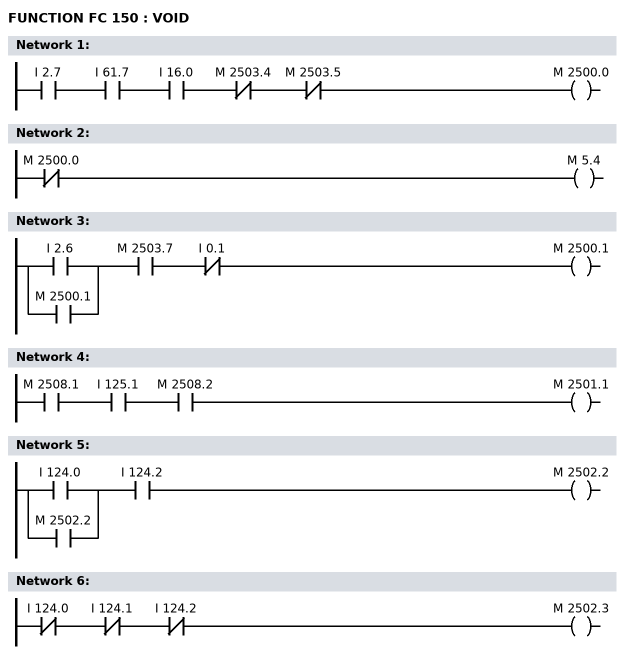

      A     I      2.7;
      A     I     61.7;
      A     I     16.0;
      AN    M   2503.4;
      AN    M   2503.5;
      =     M   2500.0;
NETWORK
TITLE =

      AN    M   2500.0;
      =     M      5.4;
NETWORK
TITLE =

      A(    ;
      O     I      2.6;
      O     M   2500.1;
      )     ;
      A     M   2503.7;
      AN    I      0.1;
      =     M   2500.1;
NETWORK
TITLE =

      A     M   2508.1;
      A     I    125.1;
      A     M   2508.2;
      =     M   2501.1;
NETWORK
TITLE =

      A(    ;
      O     I    124.0;
      O     M   2502.2;
      )     ;
      A     I    124.2;
      =     M   2502.2;
NETWORK
TITLE =

      AN    I    124.0;
      AN    I    124.1;
      AN    I    124.2;
      =     M   2502.3;
END_FUNCTION

FUNCTION_BLOCK FB 151
TITLE =
VERSION : 0.1


VAR
  S_DOWN_DL_DAECHA_CLAMP : FB 424;
  S_DOWN_DL_LIFT_LOCK : FB 424;
  S_DOWN_DL_LIFT : FB 424;
END_VAR
BEGIN
NETWORK
TITLE =
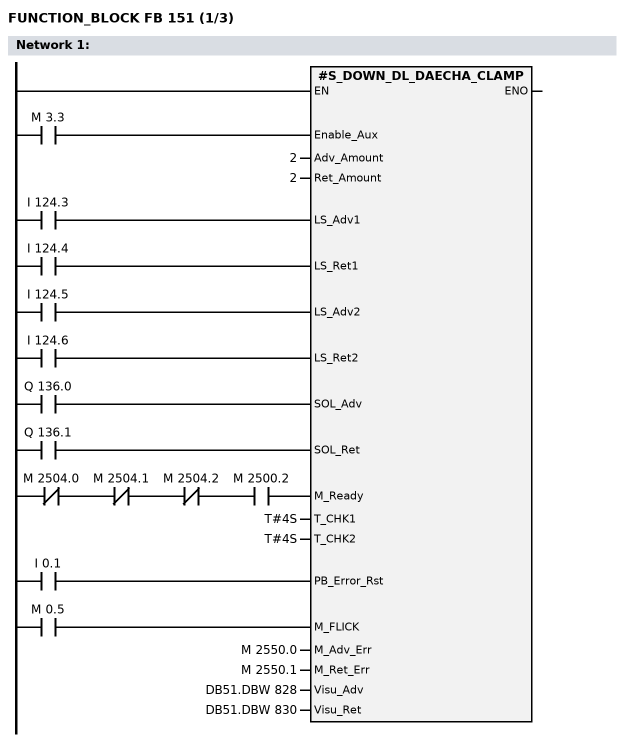

      A     M      3.3;
      =     L      0.0;
      BLD   103;
      A     I    124.3;
      =     L      0.1;
      BLD   103;
      A     I    124.4;
      =     L      0.2;
      BLD   103;
      A     I    124.5;
      =     L      0.3;
      BLD   103;
      A     I    124.6;
      =     L      0.4;
      BLD   103;
      A     Q    136.0;
      =     L      1.1;
      BLD   103;
      A     Q    136.1;
      =     L      1.2;
      BLD   103;
      AN    M   2504.0;
      AN    M   2504.1;
      AN    M   2504.2;
      A     M   2500.2;
      =     L      1.3;
      BLD   103;
      A     I      0.1;
      =     L      1.5;
      BLD   103;
      A     M      0.5;
      =     L      1.6;
      BLD   103;
      CALL #S_DOWN_DL_DAECHA_CLAMP (
           Enable_Aux               := L      0.0,
           Adv_Amount               := 2,
           Ret_Amount               := 2,
           LS_Adv1                  := L      0.1,
           LS_Ret1                  := L      0.2,
           LS_Adv2                  := L      0.3,
           LS_Ret2                  := L      0.4,
           SOL_Adv                  := L      1.1,
           SOL_Ret                  := L      1.2,
           M_Ready                  := L      1.3,
           T_CHK1                   := T#4S,
           T_CHK2                   := T#4S,
           PB_Error_Rst             := L      1.5,
           M_FLICK                  := L      1.6,
           M_Adv_Err                := M   2550.0,
           M_Ret_Err                := M   2550.1,
           Visu_Adv                 := DB51.DBW  828,
           Visu_Ret                 := DB51.DBW  830);
      NOP   0;
NETWORK
TITLE =
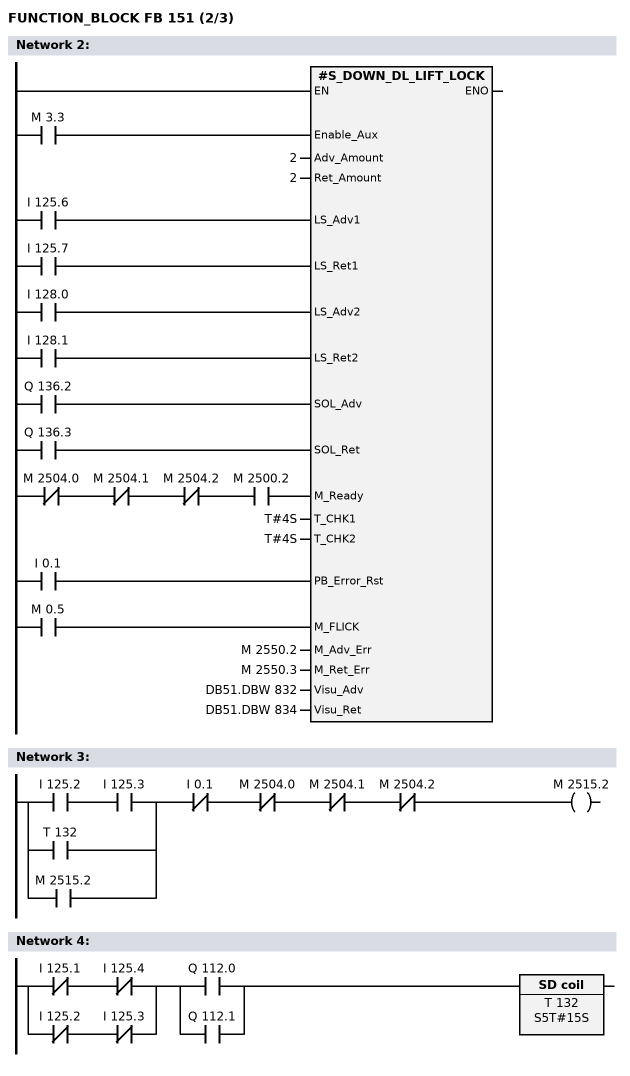

      A     M      3.3;
      =     L      0.0;
      BLD   103;
      A     I    125.6;
      =     L      0.1;
      BLD   103;
      A     I    125.7;
      =     L      0.2;
      BLD   103;
      A     I    128.0;
      =     L      0.3;
      BLD   103;
      A     I    128.1;
      =     L      0.4;
      BLD   103;
      A     Q    136.2;
      =     L      1.1;
      BLD   103;
      A     Q    136.3;
      =     L      1.2;
      BLD   103;
      AN    M   2504.0;
      AN    M   2504.1;
      AN    M   2504.2;
      A     M   2500.2;
      =     L      1.3;
      BLD   103;
      A     I      0.1;
      =     L      1.5;
      BLD   103;
      A     M      0.5;
      =     L      1.6;
      BLD   103;
      CALL #S_DOWN_DL_LIFT_LOCK (
           Enable_Aux               := L      0.0,
           Adv_Amount               := 2,
           Ret_Amount               := 2,
           LS_Adv1                  := L      0.1,
           LS_Ret1                  := L      0.2,
           LS_Adv2                  := L      0.3,
           LS_Ret2                  := L      0.4,
           SOL_Adv                  := L      1.1,
           SOL_Ret                  := L      1.2,
           M_Ready                  := L      1.3,
           T_CHK1                   := T#4S,
           T_CHK2                   := T#4S,
           PB_Error_Rst             := L      1.5,
           M_FLICK                  := L      1.6,
           M_Adv_Err                := M   2550.2,
           M_Ret_Err                := M   2550.3,
           Visu_Adv                 := DB51.DBW  832,
           Visu_Ret                 := DB51.DBW  834);
      NOP   0;
NETWORK
TITLE =

      A(    ;
      A     I    125.2;
      A     I    125.3;
      O     T    132;
      O     M   2515.2;
      )     ;
      AN    I      0.1;
      AN    M   2504.0;
      AN    M   2504.1;
      AN    M   2504.2;
      =     M   2515.2;
NETWORK
TITLE =

      A(    ;
      AN    I    125.1;
      AN    I    125.4;
      O     ;
      AN    I    125.2;
      AN    I    125.3;
      )     ;
      A(    ;
      O     Q    112.0;
      O     Q    112.1;
      )     ;
      L     S5T#15S;
      SD    T    132;
NETWORK
TITLE =
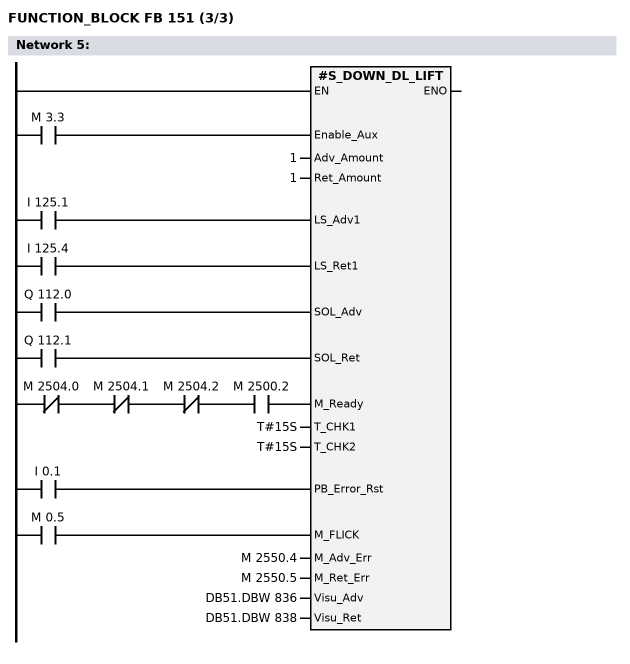

      A     M      3.3;
      =     L      0.0;
      BLD   103;
      A     I    125.1;
      =     L      0.1;
      BLD   103;
      A     I    125.4;
      =     L      0.2;
      BLD   103;
      A     Q    112.0;
      =     L      1.1;
      BLD   103;
      A     Q    112.1;
      =     L      1.2;
      BLD   103;
      AN    M   2504.0;
      AN    M   2504.1;
      AN    M   2504.2;
      A     M   2500.2;
      =     L      1.3;
      BLD   103;
      A     I      0.1;
      =     L      1.5;
      BLD   103;
      A     M      0.5;
      =     L      1.6;
      BLD   103;
      CALL #S_DOWN_DL_LIFT (
           Enable_Aux               := L      0.0,
           Adv_Amount               := 1,
           Ret_Amount               := 1,
           LS_Adv1                  := L      0.1,
           LS_Ret1                  := L      0.2,
           SOL_Adv                  := L      1.1,
           SOL_Ret                  := L      1.2,
           M_Ready                  := L      1.3,
           T_CHK1                   := T#15S,
           T_CHK2                   := T#15S,
           PB_Error_Rst             := L      1.5,
           M_FLICK                  := L      1.6,
           M_Adv_Err                := M   2550.4,
           M_Ret_Err                := M   2550.5,
           Visu_Adv                 := DB51.DBW  836,
           Visu_Ret                 := DB51.DBW  838);
      NOP   0;
END_FUNCTION_BLOCK

DATA_BLOCK DB 151
TITLE =
VERSION : 0.0

 FB 151
BEGIN
   S_DOWN_DL_DAECHA_CLAMP.Enable_Aux := FALSE;
   S_DOWN_DL_DAECHA_CLAMP.Adv_Amount := 0;
   S_DOWN_DL_DAECHA_CLAMP.Ret_Amount := 0;
   S_DOWN_DL_DAECHA_CLAMP.LS_Adv1 := FALSE;
   S_DOWN_DL_DAECHA_CLAMP.LS_Ret1 := FALSE;
   S_DOWN_DL_DAECHA_CLAMP.LS_Adv2 := FALSE;
   S_DOWN_DL_DAECHA_CLAMP.LS_Ret2 := FALSE;
   S_DOWN_DL_DAECHA_CLAMP.LS_Adv3 := FALSE;
   S_DOWN_DL_DAECHA_CLAMP.LS_Ret3 := FALSE;
   S_DOWN_DL_DAECHA_CLAMP.LS_Adv4 := FALSE;
   S_DOWN_DL_DAECHA_CLAMP.LS_Ret4 := FALSE;
   S_DOWN_DL_DAECHA_CLAMP.SOL_Adv := FALSE;
   S_DOWN_DL_DAECHA_CLAMP.SOL_Ret := FALSE;
   S_DOWN_DL_DAECHA_CLAMP.M_Ready := FALSE;
   S_DOWN_DL_DAECHA_CLAMP.T_CHK1 := T#0MS;
   S_DOWN_DL_DAECHA_CLAMP.T_CHK2 := T#0MS;
   S_DOWN_DL_DAECHA_CLAMP.PB_Lamp_CHK := FALSE;
   S_DOWN_DL_DAECHA_CLAMP.PB_Error_Rst := FALSE;
   S_DOWN_DL_DAECHA_CLAMP.M_FLICK := FALSE;
   S_DOWN_DL_DAECHA_CLAMP.M_Adv_Err := FALSE;
   S_DOWN_DL_DAECHA_CLAMP.M_Ret_Err := FALSE;
   S_DOWN_DL_DAECHA_CLAMP.LP_Adv := FALSE;
   S_DOWN_DL_DAECHA_CLAMP.LP_Ret := FALSE;
   S_DOWN_DL_DAECHA_CLAMP.Visu_Adv := W#16#0;
   S_DOWN_DL_DAECHA_CLAMP.Visu_Ret := W#16#0;
   S_DOWN_DL_DAECHA_CLAMP.Error_T1.IN := FALSE;
   S_DOWN_DL_DAECHA_CLAMP.Error_T1.PT := T#0MS;
   S_DOWN_DL_DAECHA_CLAMP.Error_T1.Q := FALSE;
   S_DOWN_DL_DAECHA_CLAMP.Error_T1.ET := T#0MS;
   S_DOWN_DL_DAECHA_CLAMP.Error_T1.STATE := B#16#0;
   S_DOWN_DL_DAECHA_CLAMP.Error_T1.STIME := T#0MS;
   S_DOWN_DL_DAECHA_CLAMP.Error_T1.ATIME := T#0MS;
   S_DOWN_DL_DAECHA_CLAMP.Error_T2.IN := FALSE;
   S_DOWN_DL_DAECHA_CLAMP.Error_T2.PT := T#0MS;
   S_DOWN_DL_DAECHA_CLAMP.Error_T2.Q := FALSE;
   S_DOWN_DL_DAECHA_CLAMP.Error_T2.ET := T#0MS;
   S_DOWN_DL_DAECHA_CLAMP.Error_T2.STATE := B#16#0;
   S_DOWN_DL_DAECHA_CLAMP.Error_T2.STIME := T#0MS;
   S_DOWN_DL_DAECHA_CLAMP.Error_T2.ATIME := T#0MS;
   S_DOWN_DL_DAECHA_CLAMP.CHK_Aux1 := FALSE;
   S_DOWN_DL_DAECHA_CLAMP.CHK_Aux2 := FALSE;
   S_DOWN_DL_DAECHA_CLAMP.Error_T1_DN := FALSE;
   S_DOWN_DL_DAECHA_CLAMP.Error_T2_DN := FALSE;
   S_DOWN_DL_DAECHA_CLAMP.Adv_Memo := FALSE;
   S_DOWN_DL_DAECHA_CLAMP.Visu_Adv_Arr[0] := FALSE;
   S_DOWN_DL_DAECHA_CLAMP.Visu_Adv_Arr[1] := FALSE;
   S_DOWN_DL_DAECHA_CLAMP.Visu_Adv_Arr[2] := FALSE;
   S_DOWN_DL_DAECHA_CLAMP.Visu_Adv_Arr[3] := FALSE;
   S_DOWN_DL_DAECHA_CLAMP.Visu_Adv_Arr[4] := FALSE;
   S_DOWN_DL_DAECHA_CLAMP.Visu_Adv_Arr[5] := FALSE;
   S_DOWN_DL_DAECHA_CLAMP.Visu_Adv_Arr[6] := FALSE;
   S_DOWN_DL_DAECHA_CLAMP.Visu_Adv_Arr[7] := FALSE;
   S_DOWN_DL_DAECHA_CLAMP.Visu_Adv_Arr[8] := FALSE;
   S_DOWN_DL_DAECHA_CLAMP.Visu_Adv_Arr[9] := FALSE;
   S_DOWN_DL_DAECHA_CLAMP.Visu_Adv_Arr[10] := FALSE;
   S_DOWN_DL_DAECHA_CLAMP.Visu_Adv_Arr[11] := FALSE;
   S_DOWN_DL_DAECHA_CLAMP.Visu_Adv_Arr[12] := FALSE;
   S_DOWN_DL_DAECHA_CLAMP.Visu_Adv_Arr[13] := FALSE;
   S_DOWN_DL_DAECHA_CLAMP.Visu_Adv_Arr[14] := FALSE;
   S_DOWN_DL_DAECHA_CLAMP.Visu_Adv_Arr[15] := FALSE;
   S_DOWN_DL_DAECHA_CLAMP.Visu_Ret_Arr[0] := FALSE;
   S_DOWN_DL_DAECHA_CLAMP.Visu_Ret_Arr[1] := FALSE;
   S_DOWN_DL_DAECHA_CLAMP.Visu_Ret_Arr[2] := FALSE;
   S_DOWN_DL_DAECHA_CLAMP.Visu_Ret_Arr[3] := FALSE;
   S_DOWN_DL_DAECHA_CLAMP.Visu_Ret_Arr[4] := FALSE;
   S_DOWN_DL_DAECHA_CLAMP.Visu_Ret_Arr[5] := FALSE;
   S_DOWN_DL_DAECHA_CLAMP.Visu_Ret_Arr[6] := FALSE;
   S_DOWN_DL_DAECHA_CLAMP.Visu_Ret_Arr[7] := FALSE;
   S_DOWN_DL_DAECHA_CLAMP.Visu_Ret_Arr[8] := FALSE;
   S_DOWN_DL_DAECHA_CLAMP.Visu_Ret_Arr[9] := FALSE;
   S_DOWN_DL_DAECHA_CLAMP.Visu_Ret_Arr[10] := FALSE;
   S_DOWN_DL_DAECHA_CLAMP.Visu_Ret_Arr[11] := FALSE;
   S_DOWN_DL_DAECHA_CLAMP.Visu_Ret_Arr[12] := FALSE;
   S_DOWN_DL_DAECHA_CLAMP.Visu_Ret_Arr[13] := FALSE;
   S_DOWN_DL_DAECHA_CLAMP.Visu_Ret_Arr[14] := FALSE;
   S_DOWN_DL_DAECHA_CLAMP.Visu_Ret_Arr[15] := FALSE;
   S_DOWN_DL_DAECHA_CLAMP.BLK_Move_Ret := 0;
   S_DOWN_DL_DAECHA_CLAMP.Enable := FALSE;
   S_DOWN_DL_DAECHA_CLAMP.Adv_End := FALSE;
   S_DOWN_DL_DAECHA_CLAMP.Ret_End := FALSE;
   S_DOWN_DL_LIFT_LOCK.Enable_Aux := FALSE;
   S_DOWN_DL_LIFT_LOCK.Adv_Amount := 0;
   S_DOWN_DL_LIFT_LOCK.Ret_Amount := 0;
   S_DOWN_DL_LIFT_LOCK.LS_Adv1 := FALSE;
   S_DOWN_DL_LIFT_LOCK.LS_Ret1 := FALSE;
   S_DOWN_DL_LIFT_LOCK.LS_Adv2 := FALSE;
   S_DOWN_DL_LIFT_LOCK.LS_Ret2 := FALSE;
   S_DOWN_DL_LIFT_LOCK.LS_Adv3 := FALSE;
   S_DOWN_DL_LIFT_LOCK.LS_Ret3 := FALSE;
   S_DOWN_DL_LIFT_LOCK.LS_Adv4 := FALSE;
   S_DOWN_DL_LIFT_LOCK.LS_Ret4 := FALSE;
   S_DOWN_DL_LIFT_LOCK.SOL_Adv := FALSE;
   S_DOWN_DL_LIFT_LOCK.SOL_Ret := FALSE;
   S_DOWN_DL_LIFT_LOCK.M_Ready := FALSE;
   S_DOWN_DL_LIFT_LOCK.T_CHK1 := T#0MS;
   S_DOWN_DL_LIFT_LOCK.T_CHK2 := T#0MS;
   S_DOWN_DL_LIFT_LOCK.PB_Lamp_CHK := FALSE;
   S_DOWN_DL_LIFT_LOCK.PB_Error_Rst := FALSE;
   S_DOWN_DL_LIFT_LOCK.M_FLICK := FALSE;
   S_DOWN_DL_LIFT_LOCK.M_Adv_Err := FALSE;
   S_DOWN_DL_LIFT_LOCK.M_Ret_Err := FALSE;
   S_DOWN_DL_LIFT_LOCK.LP_Adv := FALSE;
   S_DOWN_DL_LIFT_LOCK.LP_Ret := FALSE;
   S_DOWN_DL_LIFT_LOCK.Visu_Adv := W#16#0;
   S_DOWN_DL_LIFT_LOCK.Visu_Ret := W#16#0;
   S_DOWN_DL_LIFT_LOCK.Error_T1.IN := FALSE;
   S_DOWN_DL_LIFT_LOCK.Error_T1.PT := T#0MS;
   S_DOWN_DL_LIFT_LOCK.Error_T1.Q := FALSE;
   S_DOWN_DL_LIFT_LOCK.Error_T1.ET := T#0MS;
   S_DOWN_DL_LIFT_LOCK.Error_T1.STATE := B#16#0;
   S_DOWN_DL_LIFT_LOCK.Error_T1.STIME := T#0MS;
   S_DOWN_DL_LIFT_LOCK.Error_T1.ATIME := T#0MS;
   S_DOWN_DL_LIFT_LOCK.Error_T2.IN := FALSE;
   S_DOWN_DL_LIFT_LOCK.Error_T2.PT := T#0MS;
   S_DOWN_DL_LIFT_LOCK.Error_T2.Q := FALSE;
   S_DOWN_DL_LIFT_LOCK.Error_T2.ET := T#0MS;
   S_DOWN_DL_LIFT_LOCK.Error_T2.STATE := B#16#0;
   S_DOWN_DL_LIFT_LOCK.Error_T2.STIME := T#0MS;
   S_DOWN_DL_LIFT_LOCK.Error_T2.ATIME := T#0MS;
   S_DOWN_DL_LIFT_LOCK.CHK_Aux1 := FALSE;
   S_DOWN_DL_LIFT_LOCK.CHK_Aux2 := FALSE;
   S_DOWN_DL_LIFT_LOCK.Error_T1_DN := FALSE;
   S_DOWN_DL_LIFT_LOCK.Error_T2_DN := FALSE;
   S_DOWN_DL_LIFT_LOCK.Adv_Memo := FALSE;
   S_DOWN_DL_LIFT_LOCK.Visu_Adv_Arr[0] := FALSE;
   S_DOWN_DL_LIFT_LOCK.Visu_Adv_Arr[1] := FALSE;
   S_DOWN_DL_LIFT_LOCK.Visu_Adv_Arr[2] := FALSE;
   S_DOWN_DL_LIFT_LOCK.Visu_Adv_Arr[3] := FALSE;
   S_DOWN_DL_LIFT_LOCK.Visu_Adv_Arr[4] := FALSE;
   S_DOWN_DL_LIFT_LOCK.Visu_Adv_Arr[5] := FALSE;
   S_DOWN_DL_LIFT_LOCK.Visu_Adv_Arr[6] := FALSE;
   S_DOWN_DL_LIFT_LOCK.Visu_Adv_Arr[7] := FALSE;
   S_DOWN_DL_LIFT_LOCK.Visu_Adv_Arr[8] := FALSE;
   S_DOWN_DL_LIFT_LOCK.Visu_Adv_Arr[9] := FALSE;
   S_DOWN_DL_LIFT_LOCK.Visu_Adv_Arr[10] := FALSE;
   S_DOWN_DL_LIFT_LOCK.Visu_Adv_Arr[11] := FALSE;
   S_DOWN_DL_LIFT_LOCK.Visu_Adv_Arr[12] := FALSE;
   S_DOWN_DL_LIFT_LOCK.Visu_Adv_Arr[13] := FALSE;
   S_DOWN_DL_LIFT_LOCK.Visu_Adv_Arr[14] := FALSE;
   S_DOWN_DL_LIFT_LOCK.Visu_Adv_Arr[15] := FALSE;
   S_DOWN_DL_LIFT_LOCK.Visu_Ret_Arr[0] := FALSE;
   S_DOWN_DL_LIFT_LOCK.Visu_Ret_Arr[1] := FALSE;
   S_DOWN_DL_LIFT_LOCK.Visu_Ret_Arr[2] := FALSE;
   S_DOWN_DL_LIFT_LOCK.Visu_Ret_Arr[3] := FALSE;
   S_DOWN_DL_LIFT_LOCK.Visu_Ret_Arr[4] := FALSE;
   S_DOWN_DL_LIFT_LOCK.Visu_Ret_Arr[5] := FALSE;
   S_DOWN_DL_LIFT_LOCK.Visu_Ret_Arr[6] := FALSE;
   S_DOWN_DL_LIFT_LOCK.Visu_Ret_Arr[7] := FALSE;
   S_DOWN_DL_LIFT_LOCK.Visu_Ret_Arr[8] := FALSE;
   S_DOWN_DL_LIFT_LOCK.Visu_Ret_Arr[9] := FALSE;
   S_DOWN_DL_LIFT_LOCK.Visu_Ret_Arr[10] := FALSE;
   S_DOWN_DL_LIFT_LOCK.Visu_Ret_Arr[11] := FALSE;
   S_DOWN_DL_LIFT_LOCK.Visu_Ret_Arr[12] := FALSE;
   S_DOWN_DL_LIFT_LOCK.Visu_Ret_Arr[13] := FALSE;
   S_DOWN_DL_LIFT_LOCK.Visu_Ret_Arr[14] := FALSE;
   S_DOWN_DL_LIFT_LOCK.Visu_Ret_Arr[15] := FALSE;
   S_DOWN_DL_LIFT_LOCK.BLK_Move_Ret := 0;
   S_DOWN_DL_LIFT_LOCK.Enable := FALSE;
   S_DOWN_DL_LIFT_LOCK.Adv_End := FALSE;
   S_DOWN_DL_LIFT_LOCK.Ret_End := FALSE;
   S_DOWN_DL_LIFT.Enable_Aux := FALSE;
   S_DOWN_DL_LIFT.Adv_Amount := 0;
   S_DOWN_DL_LIFT.Ret_Amount := 0;
   S_DOWN_DL_LIFT.LS_Adv1 := FALSE;
   S_DOWN_DL_LIFT.LS_Ret1 := FALSE;
   S_DOWN_DL_LIFT.LS_Adv2 := FALSE;
   S_DOWN_DL_LIFT.LS_Ret2 := FALSE;
   S_DOWN_DL_LIFT.LS_Adv3 := FALSE;
   S_DOWN_DL_LIFT.LS_Ret3 := FALSE;
   S_DOWN_DL_LIFT.LS_Adv4 := FALSE;
   S_DOWN_DL_LIFT.LS_Ret4 := FALSE;
   S_DOWN_DL_LIFT.SOL_Adv := FALSE;
   S_DOWN_DL_LIFT.SOL_Ret := FALSE;
   S_DOWN_DL_LIFT.M_Ready := FALSE;
   S_DOWN_DL_LIFT.T_CHK1 := T#0MS;
   S_DOWN_DL_LIFT.T_CHK2 := T#0MS;
   S_DOWN_DL_LIFT.PB_Lamp_CHK := FALSE;
   S_DOWN_DL_LIFT.PB_Error_Rst := FALSE;
   S_DOWN_DL_LIFT.M_FLICK := FALSE;
   S_DOWN_DL_LIFT.M_Adv_Err := FALSE;
   S_DOWN_DL_LIFT.M_Ret_Err := FALSE;
   S_DOWN_DL_LIFT.LP_Adv := FALSE;
   S_DOWN_DL_LIFT.LP_Ret := FALSE;
   S_DOWN_DL_LIFT.Visu_Adv := W#16#0;
   S_DOWN_DL_LIFT.Visu_Ret := W#16#0;
   S_DOWN_DL_LIFT.Error_T1.IN := FALSE;
   S_DOWN_DL_LIFT.Error_T1.PT := T#0MS;
   S_DOWN_DL_LIFT.Error_T1.Q := FALSE;
   S_DOWN_DL_LIFT.Error_T1.ET := T#0MS;
   S_DOWN_DL_LIFT.Error_T1.STATE := B#16#0;
   S_DOWN_DL_LIFT.Error_T1.STIME := T#0MS;
   S_DOWN_DL_LIFT.Error_T1.ATIME := T#0MS;
   S_DOWN_DL_LIFT.Error_T2.IN := FALSE;
   S_DOWN_DL_LIFT.Error_T2.PT := T#0MS;
   S_DOWN_DL_LIFT.Error_T2.Q := FALSE;
   S_DOWN_DL_LIFT.Error_T2.ET := T#0MS;
   S_DOWN_DL_LIFT.Error_T2.STATE := B#16#0;
   S_DOWN_DL_LIFT.Error_T2.STIME := T#0MS;
   S_DOWN_DL_LIFT.Error_T2.ATIME := T#0MS;
   S_DOWN_DL_LIFT.CHK_Aux1 := FALSE;
   S_DOWN_DL_LIFT.CHK_Aux2 := FALSE;
   S_DOWN_DL_LIFT.Error_T1_DN := FALSE;
   S_DOWN_DL_LIFT.Error_T2_DN := FALSE;
   S_DOWN_DL_LIFT.Adv_Memo := FALSE;
   S_DOWN_DL_LIFT.Visu_Adv_Arr[0] := FALSE;
   S_DOWN_DL_LIFT.Visu_Adv_Arr[1] := FALSE;
   S_DOWN_DL_LIFT.Visu_Adv_Arr[2] := FALSE;
   S_DOWN_DL_LIFT.Visu_Adv_Arr[3] := FALSE;
   S_DOWN_DL_LIFT.Visu_Adv_Arr[4] := FALSE;
   S_DOWN_DL_LIFT.Visu_Adv_Arr[5] := FALSE;
   S_DOWN_DL_LIFT.Visu_Adv_Arr[6] := FALSE;
   S_DOWN_DL_LIFT.Visu_Adv_Arr[7] := FALSE;
   S_DOWN_DL_LIFT.Visu_Adv_Arr[8] := FALSE;
   S_DOWN_DL_LIFT.Visu_Adv_Arr[9] := FALSE;
   S_DOWN_DL_LIFT.Visu_Adv_Arr[10] := FALSE;
   S_DOWN_DL_LIFT.Visu_Adv_Arr[11] := FALSE;
   S_DOWN_DL_LIFT.Visu_Adv_Arr[12] := FALSE;
   S_DOWN_DL_LIFT.Visu_Adv_Arr[13] := FALSE;
   S_DOWN_DL_LIFT.Visu_Adv_Arr[14] := FALSE;
   S_DOWN_DL_LIFT.Visu_Adv_Arr[15] := FALSE;
   S_DOWN_DL_LIFT.Visu_Ret_Arr[0] := FALSE;
   S_DOWN_DL_LIFT.Visu_Ret_Arr[1] := FALSE;
   S_DOWN_DL_LIFT.Visu_Ret_Arr[2] := FALSE;
   S_DOWN_DL_LIFT.Visu_Ret_Arr[3] := FALSE;
   S_DOWN_DL_LIFT.Visu_Ret_Arr[4] := FALSE;
   S_DOWN_DL_LIFT.Visu_Ret_Arr[5] := FALSE;
   S_DOWN_DL_LIFT.Visu_Ret_Arr[6] := FALSE;
   S_DOWN_DL_LIFT.Visu_Ret_Arr[7] := FALSE;
   S_DOWN_DL_LIFT.Visu_Ret_Arr[8] := FALSE;
   S_DOWN_DL_LIFT.Visu_Ret_Arr[9] := FALSE;
   S_DOWN_DL_LIFT.Visu_Ret_Arr[10] := FALSE;
   S_DOWN_DL_LIFT.Visu_Ret_Arr[11] := FALSE;
   S_DOWN_DL_LIFT.Visu_Ret_Arr[12] := FALSE;
   S_DOWN_DL_LIFT.Visu_Ret_Arr[13] := FALSE;
   S_DOWN_DL_LIFT.Visu_Ret_Arr[14] := FALSE;
   S_DOWN_DL_LIFT.Visu_Ret_Arr[15] := FALSE;
   S_DOWN_DL_LIFT.BLK_Move_Ret := 0;
   S_DOWN_DL_LIFT.Enable := FALSE;
   S_DOWN_DL_LIFT.Adv_End := FALSE;
   S_DOWN_DL_LIFT.Ret_End := FALSE;
END_DATA_BLOCK

FUNCTION FC 151 : VOID
TITLE =
VERSION : 0.1

BEGIN
NETWORK
TITLE =
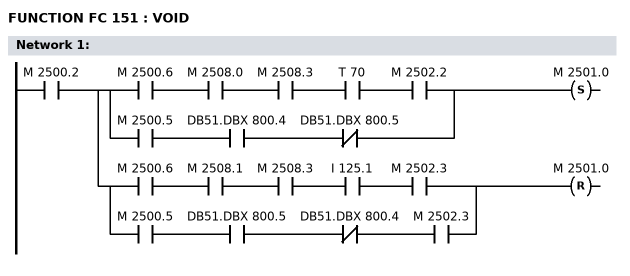

      A     M   2500.2;
      =     L      0.0;
      A     L      0.0;
      A(    ;
      A     M   2500.6;
      A     M   2508.0;
      A     M   2508.3;
      A     T     70;
      A     M   2502.2;
      O     ;
      A     M   2500.5;
      A     DB51.DBX  800.4;
      AN    DB51.DBX  800.5;
      )     ;
      S     M   2501.0;
      A     L      0.0;
      A(    ;
      A     M   2500.6;
      A     M   2508.1;
      A     M   2508.3;
      A     I    125.1;
      A     M   2502.3;
      O     ;
      A     M   2500.5;
      A     DB51.DBX  800.5;
      AN    DB51.DBX  800.4;
      A     M   2502.3;
      )     ;
      R     M   2501.0;
END_FUNCTION

FUNCTION_BLOCK FB 152
TITLE =
VERSION : 0.1

BEGIN
NETWORK
TITLE =
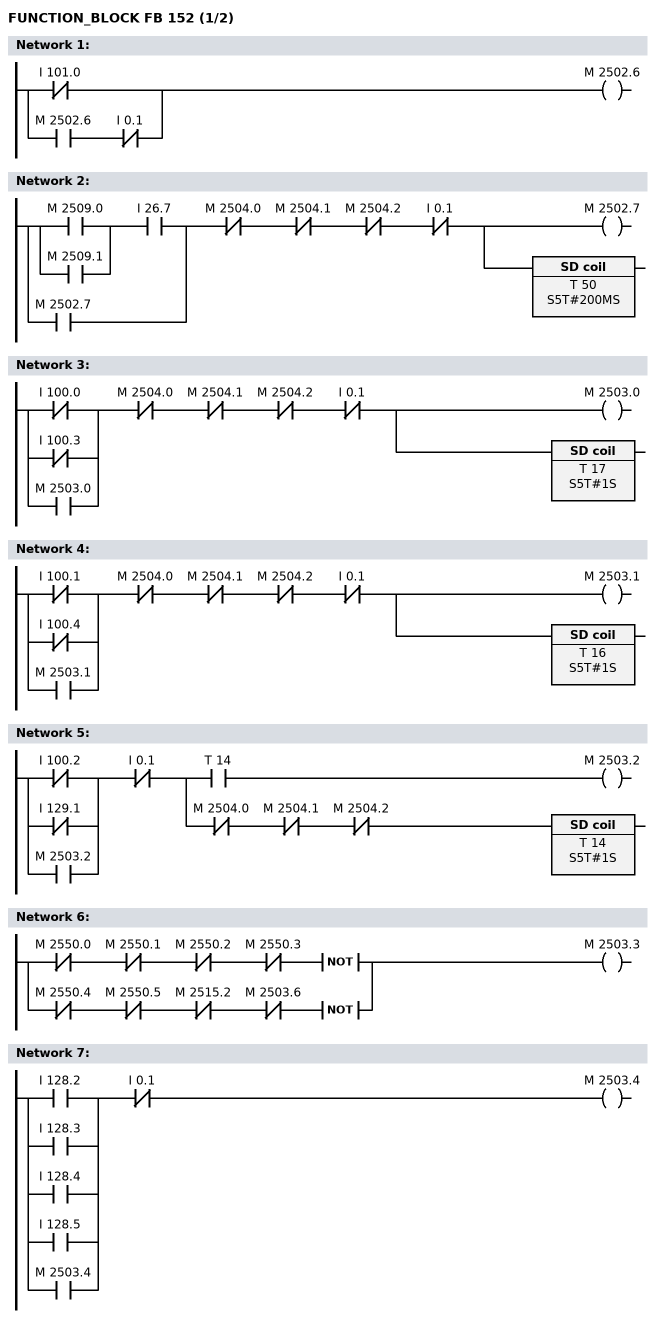

      ON    I    101.0;
      O     ;
      A     M   2502.6;
      AN    I      0.1;
      =     M   2502.6;
NETWORK
TITLE =

      A(    ;
      A(    ;
      O     M   2509.0;
      O     M   2509.1;
      )     ;
      A     I     26.7;
      O     M   2502.7;
      )     ;
      AN    M   2504.0;
      AN    M   2504.1;
      AN    M   2504.2;
      AN    I      0.1;
      =     M   2502.7;
      L     S5T#200MS;
      SD    T     50;
NETWORK
TITLE =

      A(    ;
      ON    I    100.0;
      ON    I    100.3;
      O     M   2503.0;
      )     ;
      AN    M   2504.0;
      AN    M   2504.1;
      AN    M   2504.2;
      AN    I      0.1;
      =     M   2503.0;
      L     S5T#1S;
      SD    T     17;
NETWORK
TITLE =

      A(    ;
      ON    I    100.1;
      ON    I    100.4;
      O     M   2503.1;
      )     ;
      AN    M   2504.0;
      AN    M   2504.1;
      AN    M   2504.2;
      AN    I      0.1;
      =     M   2503.1;
      L     S5T#1S;
      SD    T     16;
NETWORK
TITLE =

      A(    ;
      ON    I    100.2;
      ON    I    129.1;
      O     M   2503.2;
      )     ;
      AN    I      0.1;
      =     L      0.0;
      A     L      0.0;
      A     T     14;
      =     M   2503.2;
      A     L      0.0;
      AN    M   2504.0;
      AN    M   2504.1;
      AN    M   2504.2;
      L     S5T#1S;
      SD    T     14;
NETWORK
TITLE =

      AN    M   2550.0;
      AN    M   2550.1;
      AN    M   2550.2;
      AN    M   2550.3;
      NOT   ;
      O(    ;
      AN    M   2550.4;
      AN    M   2550.5;
      AN    M   2515.2;
      AN    M   2503.6;
      NOT   ;
      )     ;
      =     M   2503.3;
NETWORK
TITLE =

      A(    ;
      O     I    128.2;
      O     I    128.3;
      O     I    128.4;
      O     I    128.5;
      O     M   2503.4;
      )     ;
      AN    I      0.1;
      =     M   2503.4;
NETWORK
TITLE =
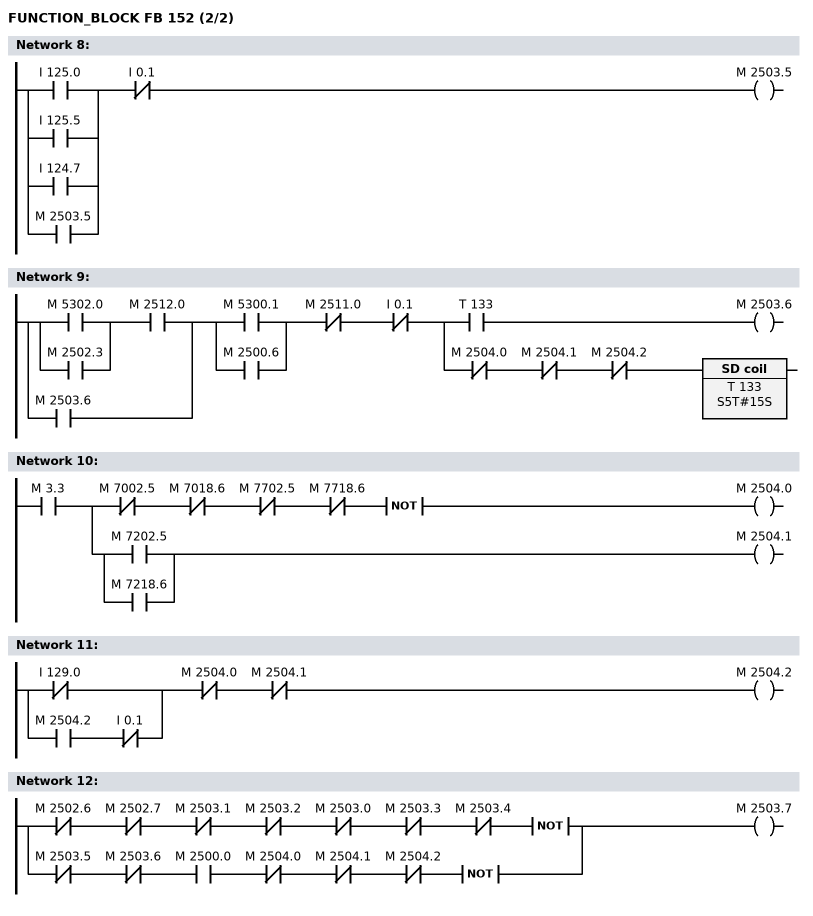

      A(    ;
      O     I    125.0;
      O     I    125.5;
      O     I    124.7;
      O     M   2503.5;
      )     ;
      AN    I      0.1;
      =     M   2503.5;
NETWORK
TITLE =

      A(    ;
      A(    ;
      O     M   5302.0;
      O     M   2502.3;
      )     ;
      A     M   2512.0;
      O     M   2503.6;
      )     ;
      A(    ;
      O     M   5300.1;
      O     M   2500.6;
      )     ;
      AN    M   2511.0;
      AN    I      0.1;
      =     L      0.0;
      A     L      0.0;
      A     T    133;
      =     M   2503.6;
      A     L      0.0;
      AN    M   2504.0;
      AN    M   2504.1;
      AN    M   2504.2;
      L     S5T#15S;
      SD    T    133;
NETWORK
TITLE =

      A     M      3.3;
      =     L      0.0;
      A     L      0.0;
      AN    M   7002.5;
      AN    M   7018.6;
      AN    M   7702.5;
      AN    M   7718.6;
      NOT   ;
      =     M   2504.0;
      A     L      0.0;
      A(    ;
      O     M   7202.5;
      O     M   7218.6;
      )     ;
      =     M   2504.1;
NETWORK
TITLE =

      A(    ;
      ON    I    129.0;
      O     ;
      A     M   2504.2;
      AN    I      0.1;
      )     ;
      AN    M   2504.0;
      AN    M   2504.1;
      =     M   2504.2;
NETWORK
TITLE =

      AN    M   2502.6;
      AN    M   2502.7;
      AN    M   2503.1;
      AN    M   2503.2;
      AN    M   2503.0;
      AN    M   2503.3;
      AN    M   2503.4;
      NOT   ;
      O(    ;
      AN    M   2503.5;
      AN    M   2503.6;
      A     M   2500.0;
      AN    M   2504.0;
      AN    M   2504.1;
      AN    M   2504.2;
      NOT   ;
      )     ;
      =     M   2503.7;
END_FUNCTION_BLOCK

DATA_BLOCK DB 152
TITLE =
VERSION : 0.0

 FB 152
BEGIN
END_DATA_BLOCK

FUNCTION FC 152 : VOID
TITLE =
VERSION : 0.1

BEGIN
NETWORK
TITLE =
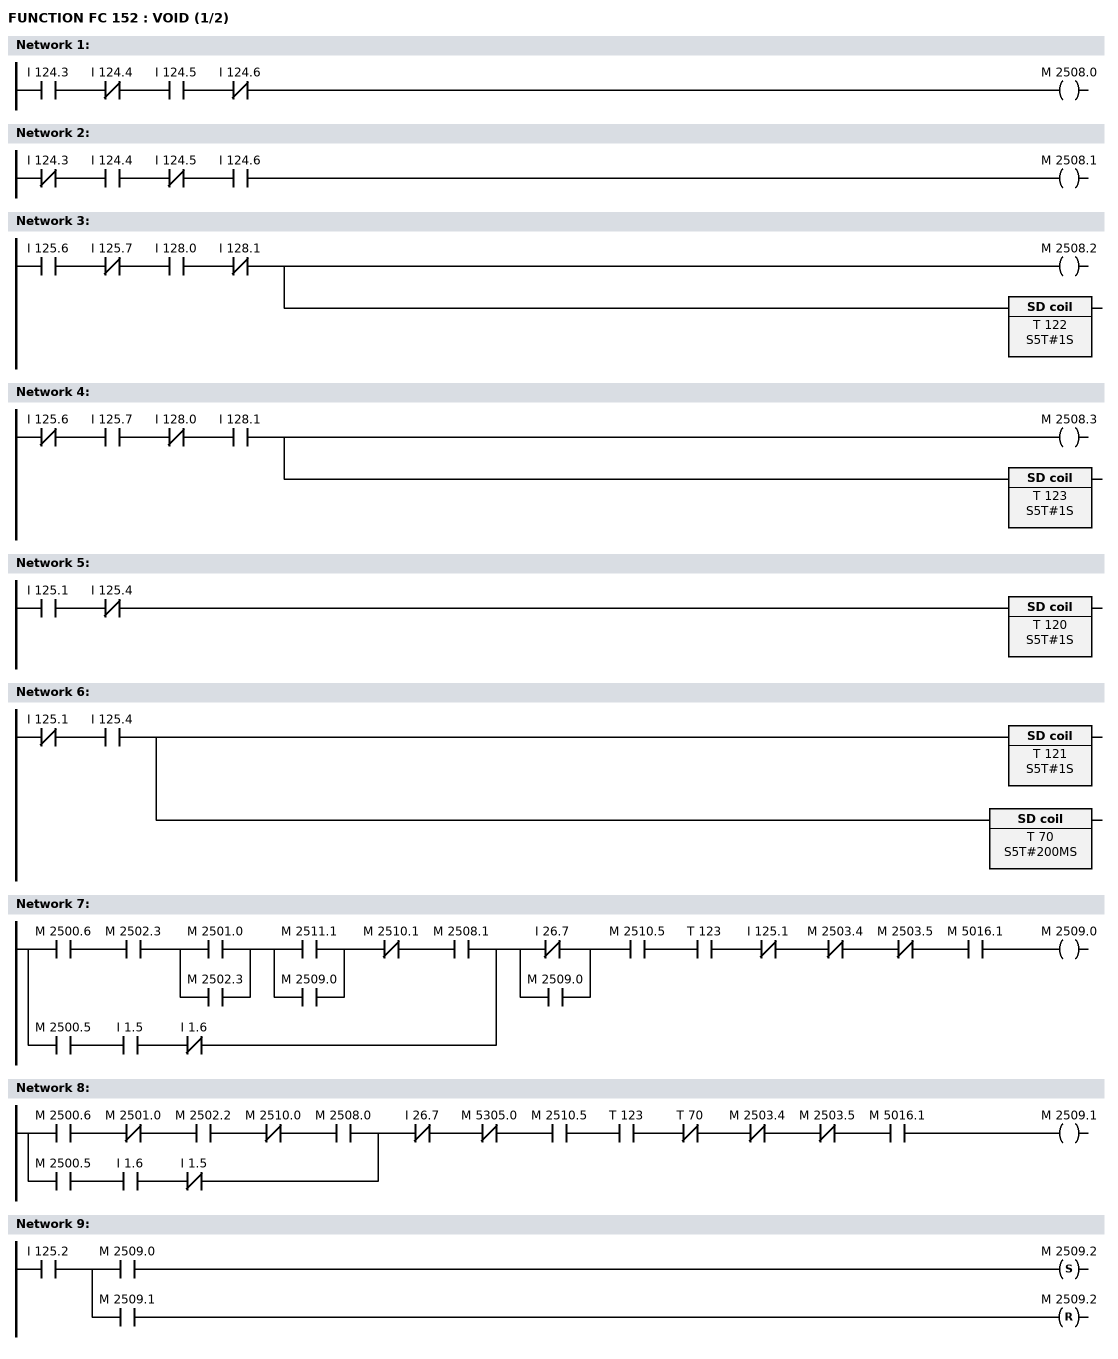

      A     I    124.3;
      AN    I    124.4;
      A     I    124.5;
      AN    I    124.6;
      =     M   2508.0;
NETWORK
TITLE =

      AN    I    124.3;
      A     I    124.4;
      AN    I    124.5;
      A     I    124.6;
      =     M   2508.1;
NETWORK
TITLE =

      A     I    125.6;
      AN    I    125.7;
      A     I    128.0;
      AN    I    128.1;
      =     M   2508.2;
      L     S5T#1S;
      SD    T    122;
NETWORK
TITLE =

      AN    I    125.6;
      A     I    125.7;
      AN    I    128.0;
      A     I    128.1;
      =     M   2508.3;
      L     S5T#1S;
      SD    T    123;
NETWORK
TITLE =

      A     I    125.1;
      AN    I    125.4;
      L     S5T#1S;
      SD    T    120;
NETWORK
TITLE =

      AN    I    125.1;
      A     I    125.4;
      L     S5T#1S;
      SD    T    121;
      L     S5T#200MS;
      SD    T     70;
NETWORK
TITLE =

      A(    ;
      A     M   2500.6;
      A     M   2502.3;
      A(    ;
      O     M   2501.0;
      O     M   2502.3;
      )     ;
      A(    ;
      O     M   2511.1;
      O     M   2509.0;
      )     ;
      AN    M   2510.1;
      A     M   2508.1;
      O     ;
      A     M   2500.5;
      A     I      1.5;
      AN    I      1.6;
      )     ;
      A(    ;
      ON    I     26.7;
      O     M   2509.0;
      )     ;
      A     M   2510.5;
      A     T    123;
      AN    I    125.1;
      AN    M   2503.4;
      AN    M   2503.5;
      A     M   5016.1;
      =     M   2509.0;
NETWORK
TITLE =

      A(    ;
      A     M   2500.6;
      AN    M   2501.0;
      A     M   2502.2;
      AN    M   2510.0;
      A     M   2508.0;
      O     ;
      A     M   2500.5;
      A     I      1.6;
      AN    I      1.5;
      )     ;
      AN    I     26.7;
      AN    M   5305.0;
      A     M   2510.5;
      A     T    123;
      AN    T     70;
      AN    M   2503.4;
      AN    M   2503.5;
      A     M   5016.1;
      =     M   2509.1;
NETWORK
TITLE =

      A     I    125.2;
      =     L      0.0;
      A     L      0.0;
      A     M   2509.0;
      S     M   2509.2;
      A     L      0.0;
      A     M   2509.1;
      R     M   2509.2;
NETWORK
TITLE =
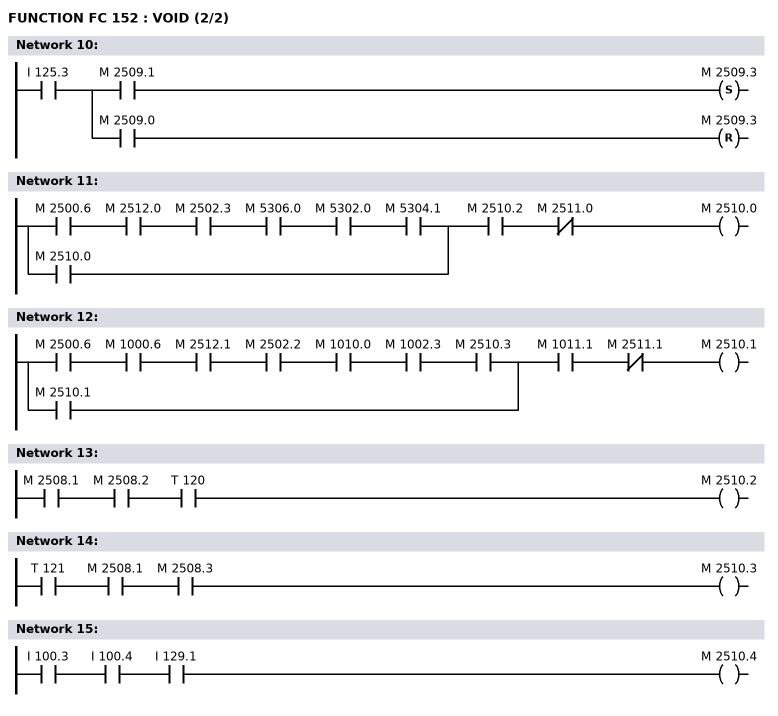

      A     I    125.3;
      =     L      0.0;
      A     L      0.0;
      A     M   2509.1;
      S     M   2509.3;
      A     L      0.0;
      A     M   2509.0;
      R     M   2509.3;
NETWORK
TITLE =

      A(    ;
      A     M   2500.6;
      A     M   2512.0;
      A     M   2502.3;
      A     M   5306.0;
      A     M   5302.0;
      A     M   5304.1;
      O     M   2510.0;
      )     ;
      A     M   2510.2;
      AN    M   2511.0;
      =     M   2510.0;
NETWORK
TITLE =

      A(    ;
      A     M   2500.6;
      A     M   1000.6;
      A     M   2512.1;
      A     M   2502.2;
      A     M   1010.0;
      A     M   1002.3;
      A     M   2510.3;
      O     M   2510.1;
      )     ;
      A     M   1011.1;
      AN    M   2511.1;
      =     M   2510.1;
NETWORK
TITLE =

      A     M   2508.1;
      A     M   2508.2;
      A     T    120;
      =     M   2510.2;
NETWORK
TITLE =

      A     T    121;
      A     M   2508.1;
      A     M   2508.3;
      =     M   2510.3;
NETWORK
TITLE =

      A     I    100.3;
      A     I    100.4;
      A     I    129.1;
      =     M   2510.4;
NETWORK
TITLE =

      AN    OV;
      =     L      0.0;
      A     L      0.0;
      A     I    100.2;
      L     S5T#500MS;
      SF    T     55;
      A     L      0.0;
      A     T     55;
      =     M   2510.6;
NETWORK
TITLE =
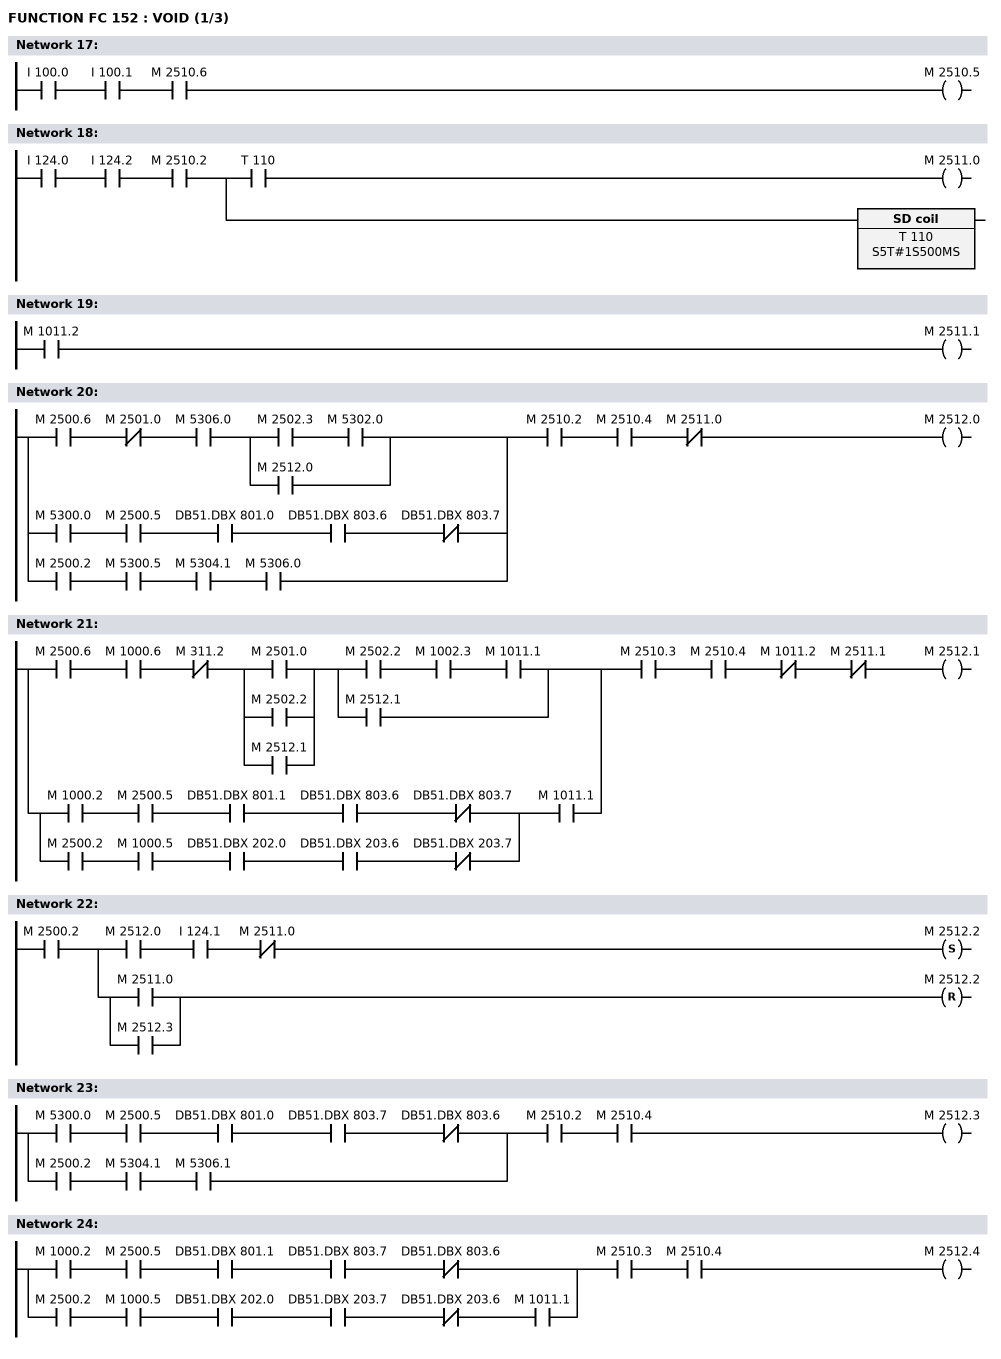

      A     I    100.0;
      A     I    100.1;
      A     M   2510.6;
      =     M   2510.5;
NETWORK
TITLE =

      A     I    124.0;
      A     I    124.2;
      A     M   2510.2;
      =     L      0.0;
      A     L      0.0;
      A     T    110;
      =     M   2511.0;
      A     L      0.0;
      BLD   102;
      L     S5T#1S500MS;
      SD    T    110;
NETWORK
TITLE =

      A     M   1011.2;
      =     M   2511.1;
NETWORK
TITLE =

      A(    ;
      A     M   2500.6;
      AN    M   2501.0;
      A     M   5306.0;
      A(    ;
      A     M   2502.3;
      A     M   5302.0;
      O     M   2512.0;
      )     ;
      O     ;
      A     M   5300.0;
      A     M   2500.5;
      A     DB51.DBX  801.0;
      A     DB51.DBX  803.6;
      AN    DB51.DBX  803.7;
      O     ;
      A     M   2500.2;
      A     M   5300.5;
      A     M   5304.1;
      A     M   5306.0;
      )     ;
      A     M   2510.2;
      A     M   2510.4;
      AN    M   2511.0;
      =     M   2512.0;
NETWORK
TITLE =

      A(    ;
      A     M   2500.6;
      A     M   1000.6;
      AN    M    311.2;
      A(    ;
      O     M   2501.0;
      O     M   2502.2;
      O     M   2512.1;
      )     ;
      A(    ;
      A     M   2502.2;
      A     M   1002.3;
      A     M   1011.1;
      O     M   2512.1;
      )     ;
      O     ;
      A(    ;
      A     M   1000.2;
      A     M   2500.5;
      A     DB51.DBX  801.1;
      A     DB51.DBX  803.6;
      AN    DB51.DBX  803.7;
      O     ;
      A     M   2500.2;
      A     M   1000.5;
      A     DB51.DBX  202.0;
      A     DB51.DBX  203.6;
      AN    DB51.DBX  203.7;
      )     ;
      A     M   1011.1;
      )     ;
      A     M   2510.3;
      A     M   2510.4;
      AN    M   1011.2;
      AN    M   2511.1;
      =     M   2512.1;
NETWORK
TITLE =

      A     M   2500.2;
      =     L      0.0;
      A     L      0.0;
      A     M   2512.0;
      A     I    124.1;
      AN    M   2511.0;
      S     M   2512.2;
      A     L      0.0;
      A(    ;
      O     M   2511.0;
      O     M   2512.3;
      )     ;
      R     M   2512.2;
NETWORK
TITLE =

      A(    ;
      A     M   5300.0;
      A     M   2500.5;
      A     DB51.DBX  801.0;
      A     DB51.DBX  803.7;
      AN    DB51.DBX  803.6;
      O     ;
      A     M   2500.2;
      A     M   5304.1;
      A     M   5306.1;
      )     ;
      A     M   2510.2;
      A     M   2510.4;
      =     M   2512.3;
NETWORK
TITLE =

      A(    ;
      A     M   1000.2;
      A     M   2500.5;
      A     DB51.DBX  801.1;
      A     DB51.DBX  803.7;
      AN    DB51.DBX  803.6;
      O     ;
      A     M   2500.2;
      A     M   1000.5;
      A     DB51.DBX  202.0;
      A     DB51.DBX  203.7;
      AN    DB51.DBX  203.6;
      A     M   1011.1;
      )     ;
      A     M   2510.3;
      A     M   2510.4;
      =     M   2512.4;
NETWORK
TITLE =
